(* CODESYS project RML AOIs.library
   Title: RML AOIs
   Version: 1.1
   Placeholder: RML AOIs
   Company: RML Toolbox

Project tree, tasks and I/O mapping:
  libraries: Tc2_Database, * (Beckhoff Automation GmbH); Tc2_Drive, * (Beckhoff Automation GmbH); Tc2_EtherCAT, * (Beckhoff Automation GmbH); Tc2_IoFunctions, * (Beckhoff Automation GmbH); Tc2_MC2, * (Beckhoff Automation GmbH); Tc2_MC2_Drive, * (Beckhoff Automation GmbH); Tc2_NCI, * (Beckhoff Automation GmbH); Tc2_Standard, * (Beckhoff Automation GmbH); Tc2_SUPS, * (Beckhoff Automation GmbH); Tc2_System, * (Beckhoff Automation GmbH); Tc2_TcpIp, * (Beckhoff Automation GmbH); Tc2_Utilities, * (Beckhoff Automation GmbH); Tc3_EventLogger, * (Beckhoff Automation GmbH); Tc3_Module, * (Beckhoff Automation GmbH); Tc2_CncHli, * (Beckhoff Automation GmbH); Tc3_CNC, * (Beckhoff Automation GmbH); Tc3_CNC_Drive, * (Beckhoff Automation GmbH)
  Objects/
    F_ImplicitChecks_V4_00/
      function F_CheckDivDint [ST]
      function F_CheckDivInt [ST]
      function F_CheckDivReal [ST]
      function F_CheckIndexBounds [ST]
      function F_CheckIndexBounds_DINT [ST]
      function F_CheckIndexBounds_REAL [ST]
      function F_CheckIndexBounds_UINT [ST]
      function F_LIMIT [ST]
    FB_AnalogueInput_V4_01/
      data type E_AInputTypeConfig
      function block FB_AnalogueInput [ST]: Alarm, AlarmMute, DebounceOff_ET, DebounceOff_PT, DebounceOn_ET, DebounceOn_PT, Description, FallingEdge, Fault, FaultTimer_ET, FaultTimer_PT, ForceOn, Input, Input2, M_AlarmMonitor, M_Alarms, M_Output, M_TypeConfig, M_UnlatchManuals, M_WarningMonitor, M_Warnings, ManOff, ManOn, ManOnQa, ManQa, Name, RisingEdge, SimInput, SimInput2, SimInputQa, StandbyReset, Value_Q, Value_Qa, Warning
    FB_AnalogueOutput_V4_01/
      data type E_AOutputTypeConfig
      function block FB_AnalogueOutput [ST]: Alarm, AlarmMute, DebounceOff_ET, DebounceOff_PT, DebounceOn_ET, DebounceOn_PT, Description, FallingEdge, Fault, FaultTimer_ET, FaultTimer_PT, ForceOn, Input, Input2, M_AlarmMonitor, M_Alarms, M_Output, M_TypeConfig, M_UnlatchManuals, M_WarningMonitor, M_Warnings, ManOff, ManOn, ManOnQa, ManQa, Name, RisingEdge, SimInput, SimInput2, SimInputQa, StandbyReset, Value_Q, Value_Qa, Warning
    FB_CNC_V1_01/
      data type E_CNC_HomingMethod
      data type E_CNC_Mode
      data type E_CNC_State
      function block FB_CNC [ST]: Alarm, AlarmMute, AutoHome, AxisEnabled, Description, Fault, FaultTimer_ET, FaultTimer_PT, FeedOverride, HandwheelSelected, Homed, M_AlarmMonitor, M_Alarms, M_AxesHandler, M_ChannelHandler, M_Homing, M_ManualMode, M_Selections, M_Spindle, M_ToolHandler, M_VariableViewer, M_WarningMonitor, M_Warnings, MachineMode, Name, ProgramEnd, ToolData, Variables, Warning
      data type ST_Handwheel
      data type ST_MachineMode
      data type ST_Position
      data type ST_Spindle
      data type ST_Tool
      data type ST_VE_CHAN0
    FB_CsvLogger_V1_01/
      function block FB_CsvLogger [ST]: Alarm, AlarmMute, Description, Enable, Fault, FaultTimer_ET, FaultTimer_PT, FB_exit, M_AlarmMonitor, M_Alarms, M_Log, M_WarningMonitor, M_Warnings, Name, Warning
    FB_Cylinder_V4_01/
      data type E_CylinderTypeConfig
      function block FB_Cylinder [ST]: Alarm, AlarmMute, AutoExtend, AutoRetract, CycleExtTime_PT, CycleRetTime_PT, Description, ExFaultTime_ET, ExFaultTime_PT, ExtendReed, ExtendReed1, ExtendSol, ForceExtend, ForceRetract, M_AlarmMonitor, M_Alarms, M_CountsReset, M_Extend, M_ExtendFault, M_ReedControl, M_ReedFault, M_Retract, M_RetractFault, M_TestCycle, M_TypeConfig, M_UnlatchManuals, M_WarningMonitor, M_Warnings, ManExtend, ManOff, ManRetract, Name, ReedFaultTime_ET, ReedFaultTime_PT, RetractReed, RetractReed1, RetractSol, RtFaultTime_ET, RtFaultTime_PT, StandbyReset, Variables, Warning
    FB_Database_V4_00/
      DUTs/
        data type ST_Example
      SQL Scripts/
        USP_Example.sql
        USP_Example_TestCall.sql
      Stored Procedures/
        function block FB_Example [ST]
      CurrentConfigDataBase.xml
      data type E_DatabaseType
      function block FB_Tc2Database [ST]: Alarm, AlarmMute, Description, M_AlarmMonitor, M_DbAlarms, M_DbServerAlarms, M_OdbcAlarms, Name
    FB_Diagnostics_V4_01/
      function block FB_Diagnostics [ST]: Alarm, AlarmMute, Description, F_DeviceState_to_String, F_LinkState_to_String, FaultTimer_PT, M_AlarmMonitor, M_AlarmReset, M_Alarms, M_CPU, M_Masters, M_Slaves, M_WarningMonitor, M_Warnings, Name, Warning
      data type ST_Diagnostics
      data type ST_MasterData
    FB_DolMotor_V4_03/
      function block FB_DolMotor [ST]: Alarm, AlarmMute, AutoFwd, AutoRev, Description, Fault, FaultTimer_PT, ForceOff, ForceOnFwd, ForceOnRev, IsolatorFeedback, M_AlarmMonitor, M_Alarms, M_MotorOutputs, M_UnlatchManuals, M_WarningMonitor, M_Warnings, ManOff, ManOnFwd, ManOnRev, ManSP1, MotorOn_ET, Name, OverloadFeedback, RunFeedback, Running, StandbyReset, StartTimer_PT, TotalMotorOnHours, TypeConfig, ValueFwd, ValueRev, Variables, Velocity, Warning
    FB_EventLogger_V4_02/
      function block FB_EventLogger [ST]: M_LogAlarm, M_LogAlert, M_LogMessage, M_LogWarning
    FB_MachineInformation_V4_00/
      function block FB_MachineInfo [ST]: M_CPU
    FB_MachinePerformance_V4_00/
      function block FB_MachinePerformance [ST]
      data type ST_Performance_SP
    FB_MiscInput_V4_02/
      data type E_InputTypeConfig
      function block FB_MiscInput [ST]: Alarm, AlarmMute, AutoStandbyReset, DebounceOff_ET, DebounceOff_PT, DebounceOn_ET, DebounceOn_PT, Description, EvaluationError, FallingEdge, Fault, FaultTimer_ET, FaultTimer_PT, ForceOn, Input, Input2, M_AlarmMonitor, M_Alarms, M_TypeConfig, M_UnlatchManuals, M_WarningMonitor, M_Warnings, ManOff, ManOn, Name, RisingEdge, SimInput, TestPulse1Fault, TestPulse2Fault, TestPulseGeneralFault, Value, Warning
    FB_MiscOutput_V4_01/
      function block FB_MiscOutput [ST]: Alarm, AlarmMute, Auto, CycleCount, Description, Fault, FaultTimer_ET, FaultTimer_PT, ForceOff, ForceOn, Input, M_AlarmMonitor, M_Alarms, M_SetOutput, M_UnlatchManuals, M_WarningMonitor, M_Warnings, ManOff, ManOn, Name, OutputOff_ET, OutputOn_ET, StandbyReset, Value, Warning
    FB_OEE_V3_01/
      function block FB_OEE [ST]
      data type ST_OEE
      data type ST_OEE_Flags_SP
      data type ST_OEE_In
      data type ST_OEE_Out
      data type ST_OEE_SP
    FB_PML_V4_01/
      function block FB_PackML [ST]: M_Administration, M_Commands, M_Indicators, M_ModeControl, M_SafetyBreach, M_StateMapping, M_StateTransitions, M_TransitionCounts
      data type ST_PMLAdmin
      data type ST_PMLControl
      data type ST_PMLData
      data type ST_PMLIndicators
      data type ST_PMLModualCommands
      data type ST_PMLState
      data type ST_PMLStatus
    FB_Service_V3_00/
      function block FB_Service [ST]
    FB_Servo_V4_07/
      Helpers/
        function F_ServoCheckWindow [ST]
        function F_ServoDirection [ST]
        function F_ServoPositionCheck [ST]
        function block FB_ServoMotionDynamics [ST]
        function block FB_ServoMove [LD]
      data type E_MoveState
      data type E_ServoMoveType
      function block FB_Servo [ST]: Alarm, AlarmMute, AutoEn, AutoHome, AxisEnabled, CamInSync, ContinuousRun, ContRun, Description, DigitalInputs, ExtControl, ExtManEn, Fault, FaultTimer_ET, FaultTimer_PT, ForceNeg, ForcePos, Homed, HomeMode, Jog, M_AlarmMonitor, M_Alarms, M_BrakeControl, M_ContinuousRun, M_ControlOutputs, M_Errors, M_GetDiagnosis, M_Homing, M_Jogging, M_MotionDynamicMove, M_MoveSuperImposed, M_MoveToPosition, M_SettingsControl, M_StateControl, M_StateOutputs, M_UnlatchManuals, M_WarningMonitor, M_Warnings, ManBrakeRelease, ManEn, ManHome, MoveDynamic, MovePos, MovePosSync, MoveSuperImpose, Moving, Name, PosDynamicOK, PosMove, PosMoveHome, PosOK, PosSyncOK, RunCam, StandStill, Unit, Variables, Warning
      data type ST_CamTable
      data type ST_ConstantVelocity_SP
      data type ST_HomePosition_SP
      data type ST_MovePosition_SP
      data type ST_MoveSuperImposed_SP
      data type ST_Settings_SP
    FB_Statistics_V4_02/
      function block FB_Statistics [ST]: CurrentRate, CycleTime, History, HistoryAvg, InstHistory, LastHour, LastMin, Reset, ThisHour, ThisMin
    FB_StepEngine_V4_03/
      function block FB_StepEngine [ST]: Alarm, AlarmMute, CurrentStep, Description, DeviceAlarm, Disable, Disabled, Fault, History, LastActiveStep, M_AlarmMonitor, M_Alarms, Name, SeqInterface, StepNum, StepReq, StepTime_ET, StepTimeDn, Variables
      data type ST_SequenceHistory
      data type ST_SequenceInterface
    FB_SystemEvent_V4_00/
      data type E_EventType
      function block FB_SystemEvent [ST]: Alarm, AlarmMute, EventTimer_ET, EventTimer_PT, Warning
    FB_TcpIpClient_V4_01/
      Example Server/
        TcpIp Sample.ivs
      data type E_ClientDataExchangeSteps
      data type E_ConnectionSteps
      function block FB_TcpIpClient [ST]: Alarm, AlarmMute, Description, Fault, FaultTimer_PT, M_AlarmMonitor, M_Alarms, M_DataExchange, M_Errors, M_MessageMonitor, M_Messages, M_WarningMonitor, M_Warnings, Name, Warning
    FB_TcpIpServer_V4_00/
      Example Client/
        EIO.cfg
        Rapid.mod
      data type E_ClientSteps
      data type E_ServerDataExchangeSteps
      data type E_ServerSteps
      function block FB_TcpIpServer [ST]: Alarm, AlarmMute, Description, Fault, FaultTimer_PT, M_AlarmMonitor, M_Alarms, M_DataExchange, M_Errors, M_MessageMonitor, M_Messages, M_RemoteClient, M_WarningMonitor, M_Warnings, Name, Warning
    FB_TimeManagement_V4_00/
      function block FB_TimeManagement [ST]: A_FirstCycle, A_LastScanTime, A_Strobes, A_SyncSystemTime, A_TimePulses, A_UpTime
      data type ST_ElapsedTime
      data type ST_TimeManagement
      data type ST_TimeManagement_SP
    FB_TwinSAFE_V4_01/
      function block FB_TwinSAFE [ST]: Alarm, Description, FaultTimer_ET, FaultTimer_PT, M_AlarmMonitor, M_Alarms, M_Control, M_WarningMonitor, M_Warnings, Name, Warning
    System_V4_01/
      data type ST_Selection
      data type ST_System
      data type ST_System_In
      data type ST_System_Out
      data type ST_System_SP
      data type ST_Variable
    text list GlobalTextList
  00000000-0000-0000-0000-000000000000|Objects\FB_Database_V4_00\SQL Scripts\USP_Example.sql
  00000000-0000-0000-0000-000000000000|Objects\FB_Database_V4_00\SQL Scripts\USP_Example_TestCall.sql
  00000000-0000-0000-0000-000000000000|Objects\FB_Database_V4_00\CurrentConfigDataBase.xml
  00000000-0000-0000-0000-000000000000|Objects\FB_TcpIpClient_V4_01\Example Server\TcpIp Sample.ivs
  00000000-0000-0000-0000-000000000000|Objects\FB_TcpIpServer_V4_00\Example Client\EIO.cfg
  00000000-0000-0000-0000-000000000000|Objects\FB_TcpIpServer_V4_00\Example Client\Rapid.mod
*)

// Objects/FB_AnalogueInput_V4_01/E_AInputTypeConfig
TYPE E_AInputTypeConfig :(
(*Type Configuration of Input*)
	eAInputType_PLC_NO				:=  0,
	eAInputType_PLC_NC 				:=  1,
	eAInputType_SAFE_NO 			:=  2,
	eAInputType_SAFE_NC				:=  3
);
END_TYPE

// Objects/FB_AnalogueOutput_V4_01/E_AOutputTypeConfig
TYPE E_AOutputTypeConfig :(
(*Type Configuration of Input*)
	eAOutputType_PLC_NO				:=  0,
	eAOutputType_PLC_NC 			:=  1,
	eAOutputType_SAFE_NO 			:=  2,
	eAOutputType_SAFE_NC			:=  3
);
END_TYPE

// Objects/FB_CNC_V1_01/E_CNC_HomingMethod
{attribute 'qualified_only'}
{attribute 'strict'}
TYPE E_CNC_HomingMethod :
(
	Homing		:=  0,
	Measurment	:=  1
)USINT;
END_TYPE

// Objects/FB_CNC_V1_01/E_CNC_Mode
TYPE E_CNC_Mode :(
		STANDBY_MODE		:=  1,
		AUTOMATIC_MODE 		:=  2,
		MDI_MODE	 		:=  3,
		MANUAL_MODE			:=  4,
		REFERENCE_MODE		:=  5
)UDINT;
END_TYPE

// Objects/FB_CNC_V1_01/E_CNC_State
TYPE E_CNC_State :(
	DESELECTED		:=  1,
	SELECTED 		:=  2,
	READY	 		:=  3,
	ACTIVE			:=  4,
	HOLD			:=  5,
	ERROR			:=  6,
	SELECTING		:=  7,
	DESELECTING		:=  8,
	PREPARING		:=  9,
	CLEARING		:=  10,
	STARTING		:=  11,
	ABORTING		:=  12,
	STOPPING		:=  13,
	RESUMING		:=  14,
	RESETTING		:=  15
)UDINT;
END_TYPE

// Objects/FB_CNC_V1_01/ST_Handwheel
TYPE ST_Handwheel :
STRUCT
	xAxisSelect		AT %I*		: BOOL;
	yAxisSelect		AT %I*		: BOOL;
	zAxisSelect		AT %I*		: BOOL;
	aAxisSelect		AT %I*		: BOOL;
	cAxisSelect		AT %I*		: BOOL;
	x10Resolution	AT %I*		: BOOL;
	x100Resolution	AT %I*		: BOOL;
	Handwheel 		AT %I*		: UINT;		//Increments for handwheel e.g. EL5101
END_STRUCT
END_TYPE

// Objects/FB_CNC_V1_01/ST_MachineMode
TYPE ST_MachineMode :
STRUCT
	/// Operation Mode 
	Standby: BOOL;
	Manual: BOOL;
	MDI: BOOL;
	Automatic: BOOL;
	Homing: BOOL;
	Select : BOOL; 
	Ready  : BOOL;
	Start: BOOL;
	Stop: BOOL;
	Reset: BOOL;
	Error: BOOL;
	Mode: UDINT;
	State: UDINT;
	/// Special functions 
	ChannelSignals: ST_ChannelSignals;
	BlockSearch: ST_BlockSearch;
	SyntaxCheck: ST_SyntaxCheck;
	ManualMode: ST_ManualMode;
	/// Strings 
	ProgramName: STRING(1024);
	MDIString: STRING(1024);
END_STRUCT
END_TYPE

// Objects/FB_CNC_V1_01/ST_Position
TYPE ST_Position :
STRUCT
	X	:	LREAL;
	Y	: 	LREAL;
	Z	: 	LREAL;
	C	: 	LREAL;
	A	: 	LREAL;
	rotX: 	LREAL;
	rotY: 	LREAL;
	rotZ: 	LREAL;
END_STRUCT
END_TYPE

// Objects/FB_CNC_V1_01/ST_Spindle
TYPE ST_Spindle :
STRUCT
	M3				: BOOL;			//Rotate Clockwise
	M4				: BOOL;			//Rotate Counter-Clockwise
	M5				: BOOL;			//Stop Spindle
	M7				: BOOL;			//Close Tool Holder
	M8				: BOOL;			//Tool Release
	M9				: BOOL;			//Tool Engage
	M19				: BOOL;			//Position Spindle (Closed-loop positioning only)
	ComVelocity		: DINT;			//Command Velocity
	ActVelocity		: LREAL;		//Actual Velocity
	Position		: DINT;			//Position Feedback
	Error			: BOOL;			//Error State
	ErrorID			: UDINT;		//Error ID
	Warm			: BOOL;			//Spindle is Warm
END_STRUCT
END_TYPE

// Objects/FB_CNC_V1_01/ST_Tool
TYPE ST_Tool :
STRUCT
	Desc	:	STRING;			// Tool Description
	Length	:	LREAL;			// Tool Length from Spindle Flange
	X		:	LREAL;			// X Location in Machine Coordinates
	Y		: 	LREAL;			// Y Location in Machine Coordinates
	Z		: 	LREAL;			// Z Location in Machine Coordinates
	SafeX	: 	LREAL;			// Safe X Location in Machine Coordinates
END_STRUCT
END_TYPE

// Objects/FB_CNC_V1_01/ST_VE_CHAN0
TYPE ST_VE_CHAN0 :
STRUCT
	Name			: STRING[127];
	Table 			: ST_Position;
	TableHeight		: LREAL;
	ParkPos 		: ST_Position;
END_STRUCT
END_TYPE

// Objects/FB_Cylinder_V4_01/E_CylinderTypeConfig
TYPE E_CylinderTypeConfig :(
(*Type Configuration of Cylinder*)
	eCylinderType_SINGLE_NORMAL			:=  0,
	eCylinderType_SINGLE_REVERSE 		:=  1,
	eCylinderType_DUEL 					:=  2
);
END_TYPE

// Objects/FB_Database_V4_00/DUTs/ST_Example
TYPE ST_Example :
STRUCT
	TimeStamp	   					:			STRING(31);//Time of Check
	UID	  							:			STRING(31);//8 Byte Unique Mac Id
	DataOk							:			STRING(31);//0=Fail, 1=Pass, 2=NA
	VisionOk						:			STRING(31);//0=Fail, 1=Pass, 2=NA
	VisionCause						:			STRING(31);//Cause of Vision Failure if Applicable
	VisionScore						: 			USINT;//0-100% Tag Find Score	
	Cycles							: 			USINT;//Amount of Cycles Through Machine
	Age	   							:			STRING(31);//Age of Tag
END_STRUCT
END_TYPE

// Objects/FB_Database_V4_00/E_DatabaseType
TYPE E_DatabaseType :(
	eMicrosoftSqlCompact				:=  0,
	eMicrosoftSql						:=  1,
	eMicrosoftAccess 					:=  2,
	eMySQL								:=  3,
	eOracle 							:=  4,
	eDB2								:=  5,
	ePostgreSQL							:=  6,
	eInterbase 							:=  7,
	eXml								:=  8,
	eAscii								:=  10
);
END_TYPE

// Objects/FB_Diagnostics_V4_01/ST_Diagnostics
TYPE ST_Diagnostics :
STRUCT
	Name					: STRING;
	ProductType				: STRING;
	CRCError				: DWORD;
	Address					: WORD;
	LinkStatus				: STRING;
	DeviceStatus			: STRING;
	NetId					: T_AmsNetId;
	LostFrames     			: UDINT;
	FramesPerSecond        	: LREAL;
	LostQueuedFrames      	: UDINT;
	QueuedFramesPerSecond 	: LREAL;
END_STRUCT
END_TYPE

// Objects/FB_Diagnostics_V4_01/ST_MasterData
TYPE ST_MasterData :
STRUCT
	ID						: WORD;
	Name					: STRING;
	Status					: STRING;
	NetId					: T_AmsNetId;
	LostFrames     			: UDINT;
	FramesPerSecond        	: LREAL;
	LostQueuedFrames      	: UDINT;
	QueuedFramesPerSecond 	: LREAL;
END_STRUCT
END_TYPE

// Objects/FB_MachinePerformance_V4_00/ST_Performance_SP
TYPE ST_Performance_SP :
STRUCT
	Current_Time							: DINT;
	Current									: ST_TIMEMANAGEMENT;
	Today_Time								: DINT;
	Today									: ST_TIMEMANAGEMENT;
	Today_Freq								: DINT;
	Today_Percent							: REAL;
	LifeTime_Time							: DINT;
	LifeTime								: ST_TIMEMANAGEMENT;
	LifeTime_Freq							: DINT;
	LifeTime_Percent						: REAL;	
END_STRUCT
END_TYPE

// Objects/FB_MiscInput_V4_02/E_InputTypeConfig
TYPE E_InputTypeConfig :(
(*Type Configuration of Input*)
	eInputType_PLC_NO				:=  0,
	eInputType_PLC_NC 				:=  1,
	eInputType_SAFE_NO 				:=  2,
	eInputType_SAFE_NC				:=  3,
	eInputType_SAFE_DUAL_NO 		:=  4,
	eInputType_SAFE_DUAL_NC 		:=  5,
	eInputType_SAFE_DUAL_NO_NC		:=  6
);
END_TYPE

// Objects/FB_OEE_V3_01/ST_OEE
TYPE ST_OEE :
STRUCT
	Inputs										: ST_OEE_In;
	Outputs										: ST_OEE_Out;
END_STRUCT
END_TYPE

// Objects/FB_OEE_V3_01/ST_OEE_Flags_SP
TYPE ST_OEE_Flags_SP :
STRUCT
	InfeedNotOK							: BOOL;				//Infeed supply below machine specification rate
	OutfeedNotOK						: BOOL;				//Dwnstreem equipment is stopping the machine from running
	GoodPiece							: BOOL;				//Good product
	RejectPiece							: BOOL;				//Reject Product
	BreakActive							: BOOL;				//Break active has been selected
	GoodPiece_Increment					: DINT;				//Good piece increment rate
	RejectPiece_Increment				: INT;				//Reject piece increment rate
	TargetProductRate					: REAL;				//Target Product Rate Per Minute
	TargetBoxRate						: REAL;				//Target Box Rate Per Minute
	BreakActive_ALM						: BOOL; 		    //Break active alarm
	InfeedTimer							: TON;				//Infeed Availability Timer
	OutfeedTimer						: TON;				//Outfeed Availability Timer
END_STRUCT
END_TYPE

// Objects/FB_OEE_V3_01/ST_OEE_In
TYPE ST_OEE_In :
STRUCT
	Sec_PulseTrigger										: BOOL;
	Break_Active											: BOOL;
	EnableIn												: BOOL;	
	Select													: BOOL;
END_STRUCT
END_TYPE

// Objects/FB_OEE_V3_01/ST_OEE_Out
TYPE ST_OEE_Out :
STRUCT
	Quality												: REAL;
	Performance											: REAL;
	Availability										: REAL;
	OEE													: REAL;
	Active												: BOOL;
	EnableOut											: BOOL;	
END_STRUCT
END_TYPE

// Objects/FB_OEE_V3_01/ST_OEE_SP
TYPE ST_OEE_SP :
STRUCT
	Start								: ST_TimeManagement;
	Stop								: ST_TimeManagement;
	Length								: ST_TimeManagement;
	Operating_Time						: ST_TimeManagement;
	Production_Time						: ST_TimeManagement;
	Break_Time							: ST_TimeManagement;
	SupplyDownTime_Time					: ST_TimeManagement;
	OutfeedDownTime_Time				: ST_TimeManagement;
	DownTime_Time						: ST_TimeManagement;			
	StartConcate						: LINT;
	StopConcate							: LINT;
	Active								: BOOL;
	ONS									: DINT;
	Operating_Seconds					: REAL;
	Production_Seconds					: REAL;
	Planned_Production					: DINT;
	StartStopConcate_Update				: BOOL;
	Break_Active						: BOOL;
	Break_Seconds						: DINT;
	TargetRate							: REAL;
	GoodPieces							: DINT;
	RejectPieces						: DINT;
	TotalPieces							: DINT;
	Availability						: REAL;
	Performance							: REAL;
	Quality								: REAL;
	OEE									: REAL;
	StateCurrent						: DINT;		
	MachinePerformance					: ARRAY[0..18] OF  ST_Performance_SP;
	SupplyDownTime_Seconds		 		: REAL;
	SupplyAvaliability					: REAL;
	OutfeedDownTime_Seconds				: REAL;
	OutfeedAvaliability					: REAL;
	DownTime_Seconds					: DINT;
	ShiftName							: STRING[22];
	RisingEdge							: BOOL;
END_STRUCT
END_TYPE

// Objects/FB_PML_V4_01/ST_PMLAdmin
TYPE ST_PMLAdmin :
STRUCT
	ModeCurrentTime				: ARRAY[0..7] OF DINT;				//Time spent in Mode
	ModeCummulativeTime			: ARRAY[0..7] OF DINT;				//Cumulative Time In Each Mode
	StateCurrentTime			: ARRAY[0..7,0..17] OF DINT;		//Value of last State Timer in each [mode].State[#]
	StateCummulativeTime		: ARRAY[0..7,0..17] OF DINT;		//Cumulative Time In Each [mode].State[#]
	ProdProcessed				: DINT;								//Number Products Processed
	DefectProd					: DINT;								//Number Defective Products
	StopReason					: DINT;								//The stop reason is the first event captured during an abort, held, suspended or stop event.
	ReworkProd					: DINT;								//Number Re-workable Products
	ResetTimerCounters			: BOOL;								//Reset timers and counters
END_STRUCT
END_TYPE

// Objects/FB_PML_V4_01/ST_PMLControl
TYPE ST_PMLControl :
STRUCT
	UnitMode					: DINT := 1;				//Unit Mode Target
	UnitModeChangeRequest		: BOOL;						//Request Unit Mode Change
	CurMachSpeed				: REAL;						//Current Machine Speed
	MatReady					: ARRAY[0..31] OF BOOL;		//Materials Ready
	MatLow						: ARRAY[0..31] OF BOOL;		//Materials Low
	State						: DINT;						//Target State
	StateChangeRequest			: BOOL;						//State Change Request
	CntrlCmd					: DINT;						//Control Command
	EquipmentInterLockBlocked 	: BOOL;						//Indicates that a downstream system is not able to accept product
	EquipmentInterLockStarved	: BOOL;						//Indicates that an upstream system is not able to supply product
END_STRUCT
END_TYPE

// Objects/FB_PML_V4_01/ST_PMLData
TYPE ST_PMLData :
STRUCT
	Control						: ST_PMLControl;						//PackML control data
	Status						: ST_PMLStatus;							//PackML status data
	Admin						: ST_PMLAdmin;							//PackML administration Data
	StateCtrl					: ST_PMLModualCommands;					//PackML state control commands
	Indicator					: ST_PMLIndicators;						//PackML interfaces
END_STRUCT
END_TYPE

// Objects/FB_PML_V4_01/ST_PMLIndicators
TYPE ST_PMLIndicators :
STRUCT
	LS_H_Output					: DINT;								//Matrix Output
	RedLamp						: BOOL;								//Red Lamp
	AmberLamp					: BOOL;								//Amber Lamp
	BlueLamp					: BOOL;								//Blue Lamp
	GreenLamp					: BOOL;								//Green Lamp
	PB_Output					: DINT;								//Matrix Output
	RedButton					: BOOL;								//Red Button 
	AmberButton					: BOOL;								//Amber Button 
	BlueButton					: BOOL;								//Blue Button 
	GreenButton					: BOOL;								//Green Button 
	Horn						: BOOL;								//Horn
END_STRUCT
END_TYPE

// Objects/FB_PML_V4_01/ST_PMLModualCommands
TYPE ST_PMLModualCommands :
STRUCT
	Cmd_Reset				: BOOL;			//Reset
	Sts_Resetting_SC		: BOOL;			//Resetting State Complete
	Cmd_Start				: BOOL;			//Start
	Sts_Starting_SC			: BOOL;			//Starting State Complete
	Cmd_Stop				: BOOL;			//Stop
	Sts_Stopping_SC			: BOOL;			//Stopping State Complete
	Cmd_Hold				: BOOL;			//Hold
	Sts_Holding_SC			: BOOL;			//Holding State Complete
	Cmd_UnHold				: BOOL;			//UnHold
	Sts_UnHolding_SC		: BOOL;			//UnHolding State Complete
	Cmd_Suspend				: BOOL;			//Suspend
	Sts_Suspending_SC		: BOOL;			//Suspending State Complete
	Cmd_UnSuspend			: BOOL;			//UnSuspend
	Sts_UnSuspending_SC		: BOOL;			//UnSuspending State Complete
	Cmd_Abort				: BOOL;			//Abort
	Sts_Aborting_SC			: BOOL;			//Aborting State Complete
	Cmd_Clear				: BOOL;			//Clear
	Sts_Clearing_SC			: BOOL;			//Clearing State Complete
	Sts_Execute_SC			: BOOL;			//Execute State Complete
	Sts_Completing_SC		: BOOL;			//Completing State Complete
END_STRUCT
END_TYPE

// Objects/FB_PML_V4_01/ST_PMLState
TYPE ST_PMLState :
STRUCT
	CurrentState		: DINT;
	Clearing			: BOOL;
	Stopped				: BOOL;
	Starting			: BOOL;
	Idle				: BOOL;
	Suspended			: BOOL;
	Execute				: BOOL;
	Stopping			: BOOL;
	Aborting			: BOOL;
	Aborted				: BOOL;
	Holding				: BOOL;
	Held				: BOOL;
	UnHolding			: BOOL;
	Suspending			: BOOL;
	UnSuspending		: BOOL;
	Resetting 			: BOOL;
	Completing			: BOOL;
	Complete			: BOOL;
END_STRUCT
END_TYPE

// Objects/FB_PML_V4_01/ST_PMLStatus
TYPE ST_PMLStatus :
STRUCT
	CommandRejected							: BOOL;							//Command Rejected
	UnitModeCurrent							: DINT;							//0 = Invalid, 1 = Production, 2 = Maintenance, 3 = Manual, 4 = Batch Production
	UnitModeRequested						: BOOL;							//Requested Unit Mode Change
	UnitModeChangeInProcess					: BOOL;							//Requested Unit Mode Change In Progress
	StateCurrent				AT	%Q*		: DINT;							//Current State Number
	StateRequested							: DINT;							//Target State
	StateChangeInProgress					: BOOL;							//State Change in Progress
	StateChangeProgress						: DINT;							//Percent Complete
	StateLastCompleted						: DINT;							//Last Completed State
	SeqNumber								: DINT;							//Pack ML Sequence Number
	CurMachspd								: DINT;							//Pack ML Current Machine Speed
	MatReady								: ARRAY[0..31] OF BOOL;			//Material Ready
	MatLow									: ARRAY[0..31] OF BOOL;			//Material Ready or Low
	MachDesignSpeed							: REAL;							//Machine Design Speed
	MachCycle								: DINT;							//Machine Cycle Count
	ProdRatio								: DINT;							//Count of primary packages per secondary package
	Dirty									: BOOL;							//Dirty indicator
	Clean									: BOOL;							//Clean indicator
	TimeToDirty								: DINT;							//Time remaining
	EquipmentAllocatedToUnitModeID			: DINT;							//Machinery Unit mode allocation
	MachineReusableForUnitModeID			: DINT;							//Resuable Unit Mode ID
	MachineReusableTimeLeft					: DINT;							//Reusable Time
	MachineStoringProductID					: DINT;							//Storing Product ID
	MachineTransferringProductID			: DINT;							//Transferring Product ID
	EquipmentInterLockBlocked 				: BOOL;							//Indicates that a downstream system is not able to accept product
	EquipmentInterLockStarved				: BOOL;							//Indicates that an upstream system is not able to supply product
END_STRUCT
END_TYPE

// Objects/FB_Servo_V4_07/E_MoveState
TYPE E_MoveState :
(
	MOVESTATE_INIT,
	MOVESTATE_ENABLE,
	MOVESTATE_FORWARD,
	MOVESTATE_BACKWARDS,
	MOVESTATE_BACKWARDSSLOW,
	MOVESTATE_NEWTARGETPOSITION,
	MOVESTATE_ERROR,
	MOVESTATE_RESET,
	MOVESTATE_CAMIN,
	MOVESTATE_SWITCHCAM,
	MOVESTATE_READCAMDATA,
	MOVESTATE_PREPARECAMMODIFICATION,
	MOVESTATE_MODIFYCAM,
	MOVESTATE_CAMSCALING,
	MOVESTATE_CAMOUT,
	MOVESTATE_STOPMASTER,
	MOVESTATE_STOPAXES
);
END_TYPE

// Objects/FB_Servo_V4_07/E_ServoMoveType
TYPE E_ServoMoveType :(
	(*Move Type Configuration of Positional Move*)
	eServoMoveType_ABSOLUTE							:=  0,
	eServoMoveType_RELATIVE 						:=  1,
	eServoMoveType_MODULO_SHORTEST_PATH 			:=  2,
	eServoMoveType_MODULO_POSITIVE 					:=  3,
	eServoMoveType_MODULO_NEGATIVE					:=  4,
	eServoMoveType_ABSOLUTE_MASTER_OFFSET 			:=  5,
	eServoMoveType_INCREMENTAL_MASTER_OFFSET		:=  6
);
END_TYPE

// Objects/FB_Servo_V4_07/ST_CamTable
TYPE ST_CamTable :
STRUCT
	TableData 		: ARRAY [0..360,0..1] OF LREAL;
	Id				: UDINT;
	Rows			: UDINT;
	Periodic		: BOOL;
	Generate		: BOOL;
	//StartMode		: MC_StartMode;
END_STRUCT
END_TYPE

// Objects/FB_Servo_V4_07/ST_ConstantVelocity_SP
TYPE ST_ConstantVelocity_SP :
STRUCT
	Direction			: MC_Direction;			//Direction of Constant Move
	Velocity			: REAL := 50;			//Velocity Value of Move
	Acceleration		: REAL := 1;			//Accleration Value of Move
	Deceleration		: REAL := 1;			//Deceleration Value of Move
	Jerk				: REAL :=25;			//Jerk Value of Move
END_STRUCT
END_TYPE

// Objects/FB_Servo_V4_07/ST_HomePosition_SP
TYPE ST_HomePosition_SP :
STRUCT
	Position			: REAL;					//Position Value to Move to
	FastVelocity		: REAL := 50;			//Fast Velocity Value of Move
	SlowVelocity		: REAL := 10;			//Slow Velocity Value of Move
	Acceleration		: REAL := 10000;		//Accleration Value of Move
	Deceleration		: REAL := 10000;		//Deceleration Value of Move
	Jerk				: REAL := 10000;		//Jerk Value of Move
	Timeout				: REAL := 5;			//Time Allowed for Move to Complete
END_STRUCT
END_TYPE

// Objects/FB_Servo_V4_07/ST_MovePosition_SP
TYPE ST_MovePosition_SP :
STRUCT
	MoveType			: E_ServoMoveType;		//Move Type Configuration of Positional Move
	Position			: REAL;					//Position Value to Move to
	Velocity			: REAL := 50;			//Velocity Value of Move
	Acceleration		: REAL := 1;			//Accleration Value of Move
	Deceleration		: REAL := 1;			//Deceleration Value of Move
	Jerk				: REAL := 25;			//Jerk Value of Move
	Timeout				: REAL := 5;			//Time Allowed for Move to Complete
END_STRUCT
END_TYPE

// Objects/FB_Servo_V4_07/ST_MoveSuperImposed_SP
TYPE ST_MoveSuperImposed_SP :
STRUCT
	Distance			: REAL;					//Relative distance to catch up or fall back with the super imposed move
	Velocity			: REAL := 50;			//Velocity Value of Move without move super imposed
	VelocityDiff		: REAL := 50;			//Velocity Value of the catch up or fall back distance
	Acceleration		: REAL := 1;			//Accleration Value of Move
	Deceleration		: REAL := 1;			//Deceleration Value of Move
	Length				: REAL;					//Length of the total move distance
END_STRUCT
END_TYPE

// Objects/FB_Servo_V4_07/ST_Settings_SP
TYPE ST_Settings_SP :
STRUCT
	HomeOffsetPosition			: LREAL;			//Home Offset Position
	HomeRequired				: BOOL;				//Used if Servo is Homed from Marker
	MaxPositionLag				: LREAL;			//Maximum Position Lag Value
	MaxPositionLagTime			: LREAL;			//Filter Time for Maximum Position Lag
	SoftPositionLimitMaxActive	: BOOL;				//Activates Soft Position Maximum Limit Monitoring
	SoftPositionLimitMinActive	: BOOL;				//Activates Soft Position Minimum Limit Monitoring
	SoftPositionLimitMax		: LREAL;			//Maximum Soft Position Limit
	SoftPositionLimitMin		: LREAL;			//Minimum Soft Position Limit
	PositionTollerance			: REAL := 1;		//Window for position OK
	ModuloFactor				: LREAL;			//Modulo (unwind) value read form drive parameters
	HomingCamSearchDirection	: BOOL;				//Direction for homing drive
	HomingSyncSearchDirection	: BOOL;				//Direction for second stage of homing
END_STRUCT
END_TYPE

// Objects/FB_StepEngine_V4_03/ST_SequenceHistory
TYPE ST_SequenceHistory :
STRUCT
	StepNum			: INT;
	StepTime		: REAL;
	Message 		: STRING; 
END_STRUCT
END_TYPE

// Objects/FB_StepEngine_V4_03/ST_SequenceInterface
TYPE ST_SequenceInterface :
STRUCT
	Held					: BOOL;
	Stopped					: BOOL;
	Reset					: BOOL;
	Suspended				: BOOL;
	Complete				: BOOL;
END_STRUCT
END_TYPE

// Objects/FB_SystemEvent_V4_00/E_EventType
TYPE E_EventType :(
	eAlarm							:=  0,
	eWarning		 				:=  1,
	eAlert		 					:=  2,
	eMessage		 				:=  3
)USINT;
END_TYPE

// Objects/FB_TcpIpClient_V4_01/E_ClientDataExchangeSteps
TYPE E_ClientDataExchangeSteps :
(
	CLIENT_DATAEXCHANGE_STATE_IDLE,
	CLIENT_DATAEXCHANGE_STATE_SEND_START,
	CLIENT_DATAEXCHANGE_STATE_SEND_WAIT,
	CLIENT_DATAEXCHANGE_STATE_RECEIVE_START,
	CLIENT_DATAEXCHANGE_STATE_RECEIVE_WAIT,
	CLIENT_DATAEXCHANGE_STATE_ERROR
);
END_TYPE

// Objects/FB_TcpIpClient_V4_01/E_ConnectionSteps
TYPE E_ConnectionSteps :
(
	CONNECTION_STATE_IDLE,
	CONNECTION_STATE_CONNECT_START,
	CONNECTION_STATE_CONNECT_WAIT,
	CONNECTION_STATE_DATAEXCHANGE_START,
	CONNECTION_STATE_DATAEXCHANGE_WAIT,
	CONNECTION_STATE_CLOSE_START,
	CONNECTION_STATE_CLOSE_WAIT,
	CONNECTION_STATE_ERROR
);
END_TYPE

// Objects/FB_TcpIpServer_V4_00/E_ClientSteps
TYPE E_ClientSteps :
(
	CLIENT_STATE_IDLE,
	CLIENT_STATE_CONNECT_START,
	CLIENT_STATE_CONNECT_WAIT,
	CLIENT_STATE_DATAEXCHANGE_START,
	CLIENT_STATE_DATAEXCHANGE_WAIT,
	CLIENT_STATE_CLOSE_START,
	CLIENT_STATE_CLOSE_WAIT,
	CLIENT_STATE_ERROR
);
END_TYPE

// Objects/FB_TcpIpServer_V4_00/E_ServerDataExchangeSteps
TYPE E_ServerDataExchangeSteps :
(
	SERVER_DATAEXCHANGE_STATE_IDLE,
	SERVER_DATAEXCHANGE_STATE_SEND_START,
	SERVER_DATAEXCHANGE_STATE_SEND_WAIT,
	SERVER_DATAEXCHANGE_STATE_RECEIVE_START,
	SERVER_DATAEXCHANGE_STATE_RECEIVE_WAIT,
	SERVER_DATAEXCHANGE_STATE_ERROR
);
END_TYPE

// Objects/FB_TcpIpServer_V4_00/E_ServerSteps
TYPE E_ServerSteps :
(
	SERVER_STATE_IDLE,
	SERVER_STATE_LISTENER_OPEN_START,
	SERVER_STATE_LISTENER_OPEN_WAIT,
	SERVER_STATE_REMOTE_CLIENTS_COMM,
	SERVER_STATE_REMOTE_CLIENTS_CLOSE,
	SERVER_STATE_LISTENER_CLOSE_START,
	SERVER_STATE_LISTENER_CLOSE_WAIT,
	SERVER_STATE_ERROR
);
END_TYPE

// Objects/FB_TimeManagement_V4_00/ST_ElapsedTime
TYPE ST_ElapsedTime :
STRUCT
	Days		: INT;
	Hours		: INT;
	Minutes		: INT;
	Seconds		: INT;
END_STRUCT
END_TYPE

// Objects/FB_TimeManagement_V4_00/ST_TimeManagement
TYPE ST_TimeManagement :
STRUCT
	CurrentTime		: TIMESTRUCT;			//Current System time
	UpTime			: ST_ElapsedTime;		//Time since last reset
	SecondPulse		: BOOL;					//On for one cycle every second
	MinutePulse		: BOOL;					//On for one cycle every minute
	HourPulse		: BOOL;					//On for one cycle every hour
	MidnightPulse	: BOOL;					//On for one cycle at Midnight
	FirstCycle		: BOOL;					//True when executing first scan
	ScanTime		: REAL;					//Last scan time (Seconds)	
	SecondsNow		: DWORD;				//Current DateTime in Seconds
	SlowFlash		: BOOL;					//Slow Flash Strobe
	FastFlash		: BOOL;					//Fast Flash Strobe
	PulseFlash		: BOOL;					//Pulse Flash Strobe
END_STRUCT
END_TYPE

// Objects/FB_TimeManagement_V4_00/ST_TimeManagement_SP
TYPE ST_TimeManagement_SP :
STRUCT
	TotalUpTime				: ST_ElapsedTime;	//Total up time of System
	PreviousDay				: INT;				//Previous day, used for midnight pulse
END_STRUCT
END_TYPE

// Objects/System_V4_01/ST_Selection
TYPE ST_Selection :
STRUCT
	Select			: BOOL;
	Queued			: BOOL;
	Enabled	    	: BOOL;
	Interlock		: BOOL;
	Messages		: STRING[255];
	Description		: STRING[255];
END_STRUCT
END_TYPE

// Objects/System_V4_01/ST_System
TYPE ST_System :
STRUCT
	Inputs					: ST_System_In;			// System inputs
	Outputs					: ST_System_Out;		// System outputs
	SystemTime				: ST_TimeManagement;	// System time and pulses	
	PackMLState				: ST_PMLState;			// System PackML data
END_STRUCT
END_TYPE

// Objects/System_V4_01/ST_System_In
TYPE ST_System_In :
STRUCT
	Start					: ST_Selection;				//Machine Start selection
	Hold					: ST_Selection;				//Machine Hold selection
	Stop					: ST_Selection;				//Machine Stop selection
	Complete				: ST_Selection;				//Machine Complete selection
	SafetyReset				: ST_Selection;				//Machine Safety Reset selection
	Reset					: ST_Selection;				//Machine Reset selection
	AlarmAck				: ST_Selection;				//Machine Alarm Acknowledge selection
	Home					: ST_Selection;				//Machine Home selection
	Simulation				: ST_Selection;				//Machine Simulation selection
	RecipeLoad				: ST_Selection;				//Operator Load Recipe Selection
	RecipeSave				: ST_Selection;				//Operator Save Recipe Selection
	RecipeChanged			: ST_Selection;				//Recipe Changed Selection
	DeleteRecipe			: ST_Selection;				//Service Reset Selection
	DoorUnlock				: ST_Selection;				//Machine Gaurd Unlock Selection
	HoursReset				: BOOL;						//Resets All Motor hours, cylinder counts, machine Hours, etc...
	AlarmMuteReset			: BOOL;						//Resets Alarm Mutes for all Alarms
	GlueStandbyReset		: BOOL;						//Resets standby for all glue machines
	Exception				: __SYSTEM.ExceptionCode;	//System Exception Handler			
END_STRUCT
END_TYPE

// Objects/System_V4_01/ST_System_Out
TYPE ST_System_Out :
STRUCT
	Energized				AT %Q*	: BOOL;					//System energized
	Energized_T1					: BOOL;					//Pneumatic soft start complete
	Energized_T2					: BOOL;					//Drives power up complete
	SafetyCellBreach				: BOOL;					//Safety cell has been breached in production state
	Alert							: BOOL;					//Machine alert active
	Alarm							: BOOL;					//Machine has an alarm active
	Warning							: BOOL;					//Machine has a warning active
	Home_EN							: BOOL;					//Machine homing is enabled
	SimulationActive				: BOOL;					//Machine simulation is active
	Energized_ET					: REAL;					//Time the system has been energized
	DeEnergized_ET					: REAL;					//Time the system has been de-energized	
	AlarmMessage					: STRING;				//Active Alarm Message
	WarningMessage					: STRING;				//Active Warning Message
	InfoMessage						: STRING;				//Active Information Message
	StatusMessage					: STRING;				//Used to display machine status on HMI
	AlertMessage					: STRING;				//Used to display alert on HMI
	RecipeSaved						: BOOL;					//Recipe Saved
	RecipeLoaded					: BOOL;					//Recipe Loaded
END_STRUCT
END_TYPE

// Objects/System_V4_01/ST_System_SP
TYPE ST_System_SP:
STRUCT
	Name					: STRING[15];			// Name for HMI
	Description				: STRING[40];			// Description for HMI
	Homed					: BOOL;					// Machine homed
	Energized_T1_PT			: REAL;					// Pneumatic soft start time
	Energized_T2_PT			: REAL;					// Drives power up time
	TimeManagement			: ST_TimeManagement_SP;	// Total up time of System
	ActiveRecipe			: STRING;				// Description of active recipe
	SelectedRecipe			: STRING;				// Description of Selected Recipe on the HMI Grid
	RecipeChanged			: BOOL;					// Recipe changed, used for operator confirmation
	ActiveRecipeIndex		: UDINT;				// Index of active recipe
END_STRUCT
END_TYPE

// Objects/System_V4_01/ST_Variable
TYPE ST_Variable :
STRUCT
	Value				:REAL;
	Description			:STRING(100);
END_STRUCT
END_TYPE

// Objects/F_ImplicitChecks_V4_00/F_CheckDivDint
FUNCTION F_CheckDivDint : DINT
VAR_INPUT
	divisor: DINT;
END_VAR

IF divisor = 0 THEN
	F_CheckDivDint:=1;
ELSE
	F_CheckDivDint:=divisor;
END_IF;

END_FUNCTION

// Objects/F_ImplicitChecks_V4_00/F_CheckDivInt
FUNCTION F_CheckDivInt : INT
VAR_INPUT
	divisor: INT;
END_VAR

IF divisor = 0 THEN
	F_CheckDivInt:=1;
ELSE
	F_CheckDivInt:=divisor;
END_IF;

END_FUNCTION

// Objects/F_ImplicitChecks_V4_00/F_CheckDivReal
FUNCTION F_CheckDivReal : REAL
VAR_INPUT
	divisor: REAL;
END_VAR

IF divisor = 0 THEN
	F_CheckDivReal:=1;
ELSE
	F_CheckDivReal:=divisor;
END_IF;

END_FUNCTION

// Objects/F_ImplicitChecks_V4_00/F_CheckIndexBounds
FUNCTION F_CheckIndexBounds : INT
VAR_INPUT
	lowerbound		: 	INT;
	upperbound		:   INT;
END_VAR
VAR_IN_OUT
	index			: 	INT;
END_VAR

IF  index < lowerbound THEN
	F_CheckIndexBounds := lowerbound;
	index 		:= lowerbound;
ELSIF  index > upperbound THEN
	F_CheckIndexBounds := upperbound;
	index 		:= upperbound;
ELSE  
	F_CheckIndexBounds := index;
END_IF

END_FUNCTION

// Objects/F_ImplicitChecks_V4_00/F_CheckIndexBounds_DINT
FUNCTION F_CheckIndexBounds_DINT : DINT
VAR_INPUT
	lowerbound		: 	DINT;
	upperbound		:   DINT;
END_VAR
VAR_IN_OUT
	index			: 	DINT;
END_VAR

IF  index < lowerbound THEN
	F_CheckIndexBounds_DINT := lowerbound;
	index 		:= lowerbound;
ELSIF  index > upperbound THEN
	F_CheckIndexBounds_DINT := upperbound;
	index 		:= upperbound;
ELSE  
	F_CheckIndexBounds_DINT := index;
END_IF

END_FUNCTION

// Objects/F_ImplicitChecks_V4_00/F_CheckIndexBounds_REAL
FUNCTION F_CheckIndexBounds_REAL : REAL
VAR_INPUT
	lowerbound		: 	REAL;
	upperbound		:   REAL;
END_VAR
VAR_IN_OUT
	index			: 	REAL;
END_VAR

IF  index < lowerbound THEN
	F_CheckIndexBounds_REAL := lowerbound;
	index 		:= lowerbound;
ELSIF  index > upperbound THEN
	F_CheckIndexBounds_REAL := upperbound;
	index 		:= upperbound;
ELSE  
	F_CheckIndexBounds_REAL := index;
END_IF

END_FUNCTION

// Objects/F_ImplicitChecks_V4_00/F_CheckIndexBounds_UINT
FUNCTION F_CheckIndexBounds_UINT : UINT
VAR_INPUT
	lowerbound		: 	UINT;
	upperbound		:   UINT;
END_VAR
VAR_IN_OUT
	index			: 	UINT;
END_VAR

IF  index < lowerbound THEN
	F_CheckIndexBounds_UINT := lowerbound;
	index 		:= lowerbound;
ELSIF  index > upperbound THEN
	F_CheckIndexBounds_UINT := upperbound;
	index 		:= upperbound;
ELSE  
	F_CheckIndexBounds_UINT := index;
END_IF

END_FUNCTION

// Objects/F_ImplicitChecks_V4_00/F_LIMIT
FUNCTION F_LIMIT : BOOL
VAR_INPUT
	En			: BOOL;
	High		: LREAL;
	Value		: LREAL;
	Low			: LREAL;
END_VAR
VAR
END_VAR

IF En = TRUE AND (Low <= High AND
 (Value >= Low AND Value <= High)) OR
 (Low >= High AND
 (Value <= Low OR Value >= High)) THEN
	F_LIMIT := TRUE;
ELSE	
	F_LIMIT := FALSE;
END_IF;

END_FUNCTION

// Objects/FB_AnalogueInput_V4_01/FB_AnalogueInput
FUNCTION_BLOCK FINAL FB_AnalogueInput EXTENDS FB_EventLogger
VAR_IN_OUT
	Control					: ST_System;
END_VAR
VAR
	_Input		AT %I*		: UINT;					//Raw Input 1 - Analogue
	_Input2		AT %I*		: BOOL;					//Raw Input 2 - Digital
	_InputLimitHigh			: REAL;					//HighHigh limit of Raw Input 1
	_InputLimitLow			: REAL;					//Low limit of Raw Input 1
	_InputLimitHighHigh		: REAL;					//HighHigh limit of Raw Input 1
	_InputLimitLowLow		: REAL;					//LowLow limit of Raw Input 1
	_ManOnQa				: BOOL;					//Manual On Analogue Input
	_ManQa					: REAL;					//Manual Analogue Input
	_ManOn					: BOOL;					//Manual On
	_ManOff					: BOOL;					//Manual Off
	_ForceOn				: BOOL;					//Force On
	_ForceOff				: BOOL;					//Force Off
	_Fault					: BOOL;					//Fault
	_SimInput				: BOOL;		        	//Simulates Analogue Input
	_SimInput2				: BOOL;					//Simulates Digital Input
	_SimInputQa				: REAL;					//Value of Simulated Analogue Input
	_Value_Q	AT %Q*		: BOOL;					//Value of Input - Digital
	_Value_Qa	AT %Q*		: REAL;					//Value of Input - Analogue
	_FallingEdge			: BOOL;					//Falling Edge of Value Signal
	_RisingEdge				: BOOL;					//Raising Edge of Value Signal
	_DebounceOn_ET			: REAL;					//Debounce On Elapsed Time
	_DebounceOff_ET			: REAL;					//Debounce Off Elapsed Time
	_FaultTimer_ET			: REAL;					//Fault timer elapsed
	_Alarm					: BOOL;					//Device Alarm
	_Warning				: BOOL;					//Device Warning
	_AlarmNum				: DINT;					//Device Alarm Number
	_WarningNum				: DINT;					//Device Warning Number
	_riseEdge				: R_TRIG;				//Rising Edge Value Trigger
	_fallEdge				: F_TRIG;				//Falling Edge Value Trigger
	_Scale_Max				: REAL;					//Current Maximum (mA)
	_Scale_Min				: REAL;					//Current minimum (mA)
	_Scale_Value			: REAL;					//Current Value (mA)
	_Bit_Value				: REAL;					//Analogue Value Input
	_Bit_Max				: REAL;					//Maximum Bit Value (typically 32767)
	_Bit_Min				: REAL;					//Minimum Bit Value (typically 0)
	_Physical_Min			: REAL;					//Minimum Physical Value
	_Physical_Max			: REAL;					//Maximum Physical Value
	_ConfInput				: BOOL;					//Confirgured Input
	_DebounceOn_DN			: BOOL;					//Debounce On Timer is Done
	_DebounceOff_DN			: BOOL;					//Debounce Off Timer is Done
	_R_Trig					: ARRAY[0..9] OF R_TRIG;//Private Rising Edge Triggers
END_VAR
VAR PERSISTENT
	_Name					: STRING[15];			//Name for HMI
	_Description			: STRING[40];			//Description for HMI
	_AlarmMute				: BOOL;					//Alarm Mute
	_TypeConfig				: E_AInputTypeConfig;	//Type congifuration
	_DebounceOn_PT			: REAL;					//Debounce on timer preset time
	_DebounceOff_PT			: REAL;					//Debounce off timer preset time
	_FaultTimer_PT			: REAL;					//Fault timer preset time
	_HighAlarmLimit			: BOOL;					//Input Value is approaching the maximum operating limit.
	_LowAlarmLimit			: BOOL;					//Input Value is approaching the minimum operating limit.
	_HighHighAlarmLimit		: BOOL;					//Input Value is above  the maximum operating limit
	_LowLowAlarmLimit		: BOOL;					//Input Value is below the minimum operating limit.
	_BitValue_Max			: INT;					//Maximum Bit Value (typically 32767)
	_BitValue_Min			: INT;					//Minimum Bit Value (typically 0)
	_PhysicalValue_Min		: INT;					//Minimum Physical Value
	_PhysicalValue_Max		: INT;					//Maximum Physical Value
	_ScaleValue_Min			: INT;					//Minimum Scale Value				
	_ScaleValue_Max			: INT;					//Maximum Scale Value
END_VAR

M_TypeConfig();
M_AlarmMonitor();
M_WarningMonitor();
M_UnlatchManuals();
M_Output();

//Debounce On Timer
IF _ConfInput = TRUE AND NOT _ForceOff AND NOT _ManOff THEN
	_DebounceOn_ET := _DebounceOn_ET + Control.SystemTime.ScanTime;
	_debounceOn_DN := _DebounceOn_ET > _DebounceOn_PT;
ELSE
	_debounceOn_DN := FALSE;
END_IF
IF _debounceOn_DN OR _ForceOn OR _ManOn THEN
	_Value_Q := TRUE;
	_DebounceOff_ET := 0;
END_IF

//Debounce Off Timer
IF _ConfInput = FALSE AND NOT _ForceOn AND NOT _ManOn THEN
	_DebounceOff_ET := _DebounceOff_ET + Control.SystemTime.ScanTime;
	_debounceOff_DN := _DebounceOff_ET > _DebounceOff_PT;
ELSE
	_debounceOff_DN := FALSE;
END_IF
IF _debounceOff_DN OR _ForceOff OR _ManOff THEN
	_Value_Q:= FALSE;
	_DebounceOn_ET := 0;
END_IF

//Rising Edge Trigger 
_riseEdge(CLK := _Value_Q);
_RisingEdge := _riseEdge.Q;

//Falling Edge Trigger
_fallEdge(CLK := _Value_Q);
_FallingEdge := _fallEdge.Q;

{attribute 'monitoring' := 'variable'}
PROPERTY PUBLIC Alarm : Bool
GET
Alarm := _Alarm;
END_GET
END_PROPERTY

{attribute 'monitoring' := 'variable'}
PROPERTY PUBLIC AlarmMute : BOOL
SET
AlarmMute := _AlarmMute;
END_SET
END_PROPERTY

{attribute 'monitoring' := 'variable'}
PROPERTY PUBLIC DebounceOff_ET : real
GET
DebounceOff_ET := _DebounceOff_ET;
END_GET
END_PROPERTY

{attribute 'monitoring' := 'variable'}
PROPERTY PUBLIC DebounceOff_PT : real
GET
DebounceOff_PT := _DebounceOff_PT;
END_GET
SET
_DebounceOff_PT := DebounceOff_PT;
END_SET
END_PROPERTY

{attribute 'monitoring' := 'variable'}
PROPERTY PUBLIC DebounceOn_ET : real
GET
DebounceOn_ET := _DebounceOn_ET;
END_GET
END_PROPERTY

{attribute 'monitoring' := 'variable'}
PROPERTY PUBLIC DebounceOn_PT : real
GET
DebounceOn_PT := _DebounceOn_PT;
END_GET
SET
_DebounceOn_PT := DebounceOn_PT;
END_SET
END_PROPERTY

{attribute 'monitoring' := 'variable'}
PROPERTY PUBLIC Description : String[40]
GET
Description := _Description;
END_GET
SET
_Description := Description;
END_SET
END_PROPERTY

{attribute 'monitoring' := 'variable'}
PROPERTY PUBLIC FallingEdge : Bool
GET
FallingEdge := _FallingEdge;
END_GET
END_PROPERTY

{attribute 'monitoring' := 'variable'}
PROPERTY PUBLIC Fault : Bool
SET
_Fault := Fault;
END_SET
END_PROPERTY

{attribute 'monitoring' := 'variable'}
PROPERTY PUBLIC FaultTimer_ET : real
GET
FaultTimer_ET := _FaultTimer_ET;
END_GET
END_PROPERTY

{attribute 'monitoring' := 'variable'}
PROPERTY PUBLIC FaultTimer_PT : real
GET
FaultTimer_PT := _FaultTimer_PT;
END_GET
SET
_FaultTimer_PT := FaultTimer_PT;
END_SET
END_PROPERTY

{attribute 'monitoring' := 'variable'}
PROPERTY PUBLIC ForceOn : Bool
GET
ForceOn := _ForceOn;
END_GET
SET
_ForceOn := ForceOn;
END_SET
END_PROPERTY

{attribute 'monitoring' := 'variable'}
PROPERTY PUBLIC Input : UINT
GET
Input := _Input;
END_GET
END_PROPERTY

{attribute 'monitoring' := 'variable'}
PROPERTY PUBLIC Input2 : Bool
GET
Input2 := _Input2;
END_GET
END_PROPERTY

METHOD PRIVATE M_AlarmMonitor
VAR_INPUT
END_VAR
VAR_INST
END_VAR
VAR_INST // added by the converter: edge detectors and wires of the graphical bodies
    _w1, _w2, _w3, _w4, _w5 : BOOL;
    _rt1 : R_TRIG;
END_VAR
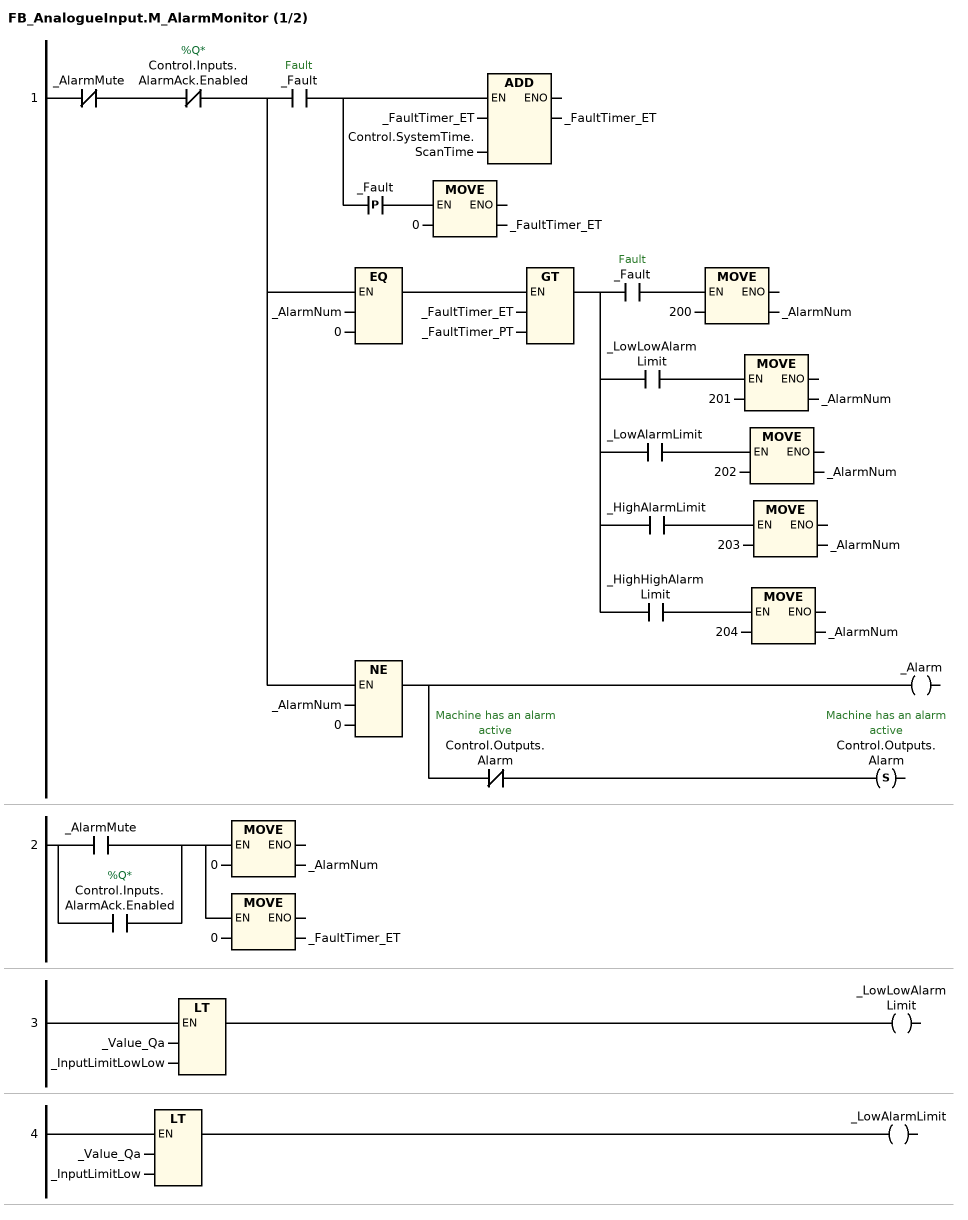
// NETWORK 1
//   Control.Inputs.AlarmAck.Enabled: AT %Q*
//   _Fault: Fault
//   _FaultTimer_ET: Fault timer elapsed
//   Control.SystemTime.ScanTime: Last scan time (Seconds)
//   _FaultTimer_PT: Fault timer preset time
//   Control.Outputs.Alarm: Machine has an alarm active
_w1 := NOT _AlarmMute AND NOT Control.Inputs.AlarmAck.Enabled;
_w2 := _w1 AND _Fault;
IF _w2 THEN _FaultTimer_ET := _FaultTimer_ET + Control.SystemTime.ScanTime; END_IF
_rt1(CLK := _Fault);
IF _w2 AND _rt1.Q THEN _FaultTimer_ET := 0; END_IF
_w3 := _w1 AND _AlarmNum = 0 AND _FaultTimer_ET > _FaultTimer_PT;
IF _w3 AND _Fault THEN _AlarmNum := 200; END_IF
IF _w3 AND _LowLowAlarmLimit THEN _AlarmNum := 201; END_IF
IF _w3 AND _LowAlarmLimit THEN _AlarmNum := 202; END_IF
IF _w3 AND _HighAlarmLimit THEN _AlarmNum := 203; END_IF
IF _w3 AND _HighHighAlarmLimit THEN _AlarmNum := 204; END_IF
_w4 := _w1 AND _AlarmNum <> 0;
_Alarm := _w4;
Control.Outputs.Alarm S= _w4 AND NOT Control.Outputs.Alarm;

// NETWORK 2
//   Control.Inputs.AlarmAck.Enabled: AT %Q*
//   _FaultTimer_ET: Fault timer elapsed
_w5 := _AlarmMute OR Control.Inputs.AlarmAck.Enabled;
IF _w5 THEN _AlarmNum := 0; END_IF
IF _w5 THEN _FaultTimer_ET := 0; END_IF

// NETWORK 3
_LowLowAlarmLimit := _Value_Qa < _InputLimitLowLow;

// NETWORK 4
_LowAlarmLimit := _Value_Qa < _InputLimitLow;

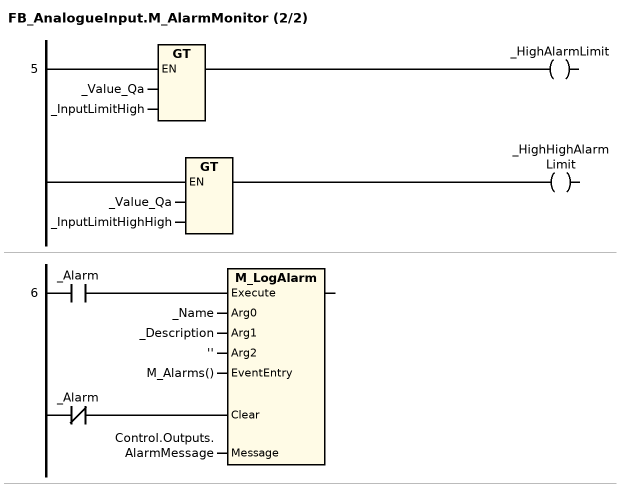
// NETWORK 5
_HighAlarmLimit := _Value_Qa > _InputLimitHigh;
_HighHighAlarmLimit := _Value_Qa > _InputLimitHighHigh;

// NETWORK 6
M_LogAlarm(Execute := _Alarm, Arg0 := _Name, Arg1 := _Description, Arg2 := '', EventEntry := M_Alarms(), Clear := NOT _Alarm, Message := Control.Outputs.AlarmMessage);
END_METHOD

METHOD PRIVATE M_Alarms : TcEventEntry
VAR_INPUT
END_VAR
CASE _AlarmNum OF
	201: M_Alarms:= TC_Events.TcAnalogueInput.A_201;//Low Low Limit Alarm
	202: M_Alarms:= TC_Events.TcAnalogueInput.A_202;//Low Limit Alarm			
	203: M_Alarms:= TC_Events.TcAnalogueInput.A_203;//High Limit Alarm
	204: M_Alarms:= TC_Events.TcAnalogueInput.A_204;//High High Limit Alarm							
ELSE
	M_Alarms:= TC_Events.TcAnalogueInput.A_Undefined;
END_CASE
END_METHOD

METHOD PRIVATE M_Output
VAR
END_VAR
VAR_INST
END_VAR
// Convert UINTs to INTs
_Scale_Min := ANY_TO_REAL(_ScaleValue_Min);
_Scale_Max := ANY_TO_REAL(_ScaleValue_Max);
_Bit_Value := ANY_TO_REAL(_Input);
_Bit_Max := ANY_TO_REAL(_BitValue_Max);		
_Bit_Min := ANY_TO_REAL(_BitValue_Min);		
_Physical_Min := ANY_TO_REAL(_PhysicalValue_Min);
_Physical_Max := ANY_TO_REAL(_PhysicalValue_Max);

IF _ManOnQa THEN
	_Value_Qa := _ManQa;
ELSIF _SimInput THEN
	_Value_Qa := _SimInputQa;
ELSIF _BitValue_Max <> 0 AND _PhysicalValue_Max <> 0 AND _ScaleValue_Max <> 0 THEN	
	// Calculate present electrical current value
	_Scale_Value := (((_Scale_Max - _Scale_Min)/F_CheckDivReal(divisor:=(_Bit_max - _Bit_min))) * (_Bit_Value - _Bit_min)) + _Scale_Min;

	// Convert electrical current value into measurable units
	_Value_Qa := (((_Physical_Max - _Physical_Min)/F_CheckDivReal(divisor:=(_Scale_Max - _Scale_Min))) * (_Scale_Value - _Scale_Min)) + _Physical_Min;	
END_IF
END_METHOD

METHOD PRIVATE M_TypeConfig
VAR_INPUT
END_VAR
VAR_INST
END_VAR
CASE _TypeConfig OF
	eAInputType_PLC_NO, eAInputType_SAFE_NO : 
		IF _Input2 OR _SimInput2 THEN
			_ConfInput := TRUE;
		ELSE
			_ConfInput := FALSE;
		END_IF
	eAInputType_PLC_NC, eAInputType_SAFE_NC : 
		IF NOT _Input2 OR _SimInput2 THEN
			_ConfInput := TRUE;
		ELSE
			_ConfInput := FALSE;
		END_IF
END_CASE
END_METHOD

METHOD PRIVATE M_UnlatchManuals
VAR_INPUT
END_VAR
VAR_INST
END_VAR
VAR_INST // added by the converter: edge detectors and wires of the graphical bodies
    _rt1, _rt2, _rt3 : R_TRIG;
END_VAR
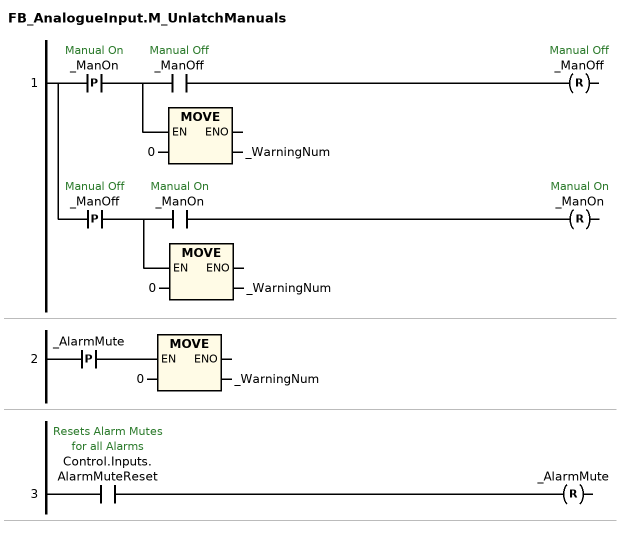
// NETWORK 1
//   _ManOn: Manual On
//   _ManOff: Manual Off
_rt1(CLK := _ManOn);
_ManOff R= _rt1.Q AND _ManOff;
IF _rt1.Q THEN _WarningNum := 0; END_IF
_rt2(CLK := _ManOff);
_ManOn R= _rt2.Q AND _ManOn;
IF _rt2.Q THEN _WarningNum := 0; END_IF

// NETWORK 2
_rt3(CLK := _AlarmMute);
IF _rt3.Q THEN _WarningNum := 0; END_IF

// NETWORK 3
//   Control.Inputs.AlarmMuteReset: Resets Alarm Mutes for all Alarms
_AlarmMute R= Control.Inputs.AlarmMuteReset;
END_METHOD

METHOD PRIVATE M_WarningMonitor
VAR_INPUT
END_VAR
VAR_INST
END_VAR
VAR_INST // added by the converter: edge detectors and wires of the graphical bodies
    _w1 : BOOL;
END_VAR
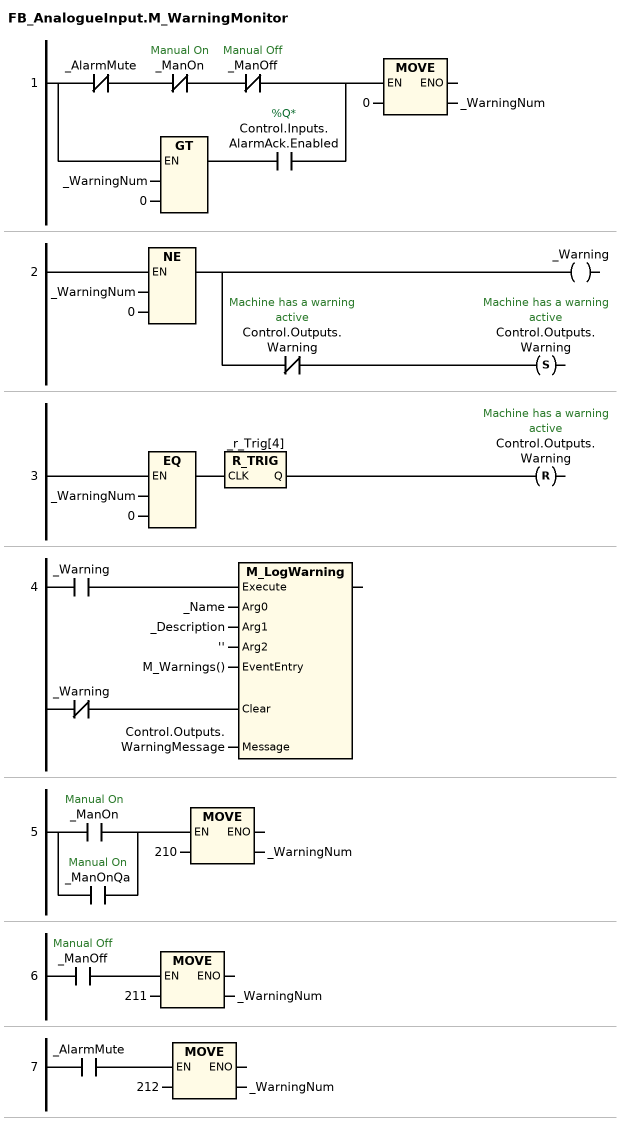
// NETWORK 1
//   _ManOn: Manual On
//   _ManOff: Manual Off
//   Control.Inputs.AlarmAck.Enabled: AT %Q*
IF NOT _AlarmMute AND NOT _ManOn AND NOT _ManOff OR _WarningNum > 0 AND Control.Inputs.AlarmAck.Enabled THEN
    _WarningNum := 0;
END_IF

// NETWORK 2
//   Control.Outputs.Warning: Machine has a warning active
_w1 := _WarningNum <> 0;
_Warning := _w1;
Control.Outputs.Warning S= _w1 AND NOT Control.Outputs.Warning;

// NETWORK 3
//   Control.Outputs.Warning: Machine has a warning active
_r_Trig[4](CLK := _WarningNum = 0); // R_TRIG
Control.Outputs.Warning R= _r_Trig[4].Q;

// NETWORK 4
M_LogWarning(Execute := _Warning, Arg0 := _Name, Arg1 := _Description, Arg2 := '', EventEntry := M_Warnings(), Clear := NOT _Warning, Message := Control.Outputs.WarningMessage);

// NETWORK 5
//   _ManOn: Manual On
//   _ManOnQa: Manual On
IF _ManOn OR _ManOnQa THEN _WarningNum := 210; END_IF

// NETWORK 6
//   _ManOff: Manual Off
IF _ManOff THEN _WarningNum := 211; END_IF

// NETWORK 7
IF _AlarmMute THEN _WarningNum := 212; END_IF
END_METHOD

METHOD PRIVATE M_Warnings : TcEventEntry
VAR_INPUT
END_VAR
CASE _WarningNum OF
	210: M_Warnings:= TC_Events.TcAnalogueInput.W_210;//Manual ON Enabled
	211: M_Warnings:= TC_Events.TcAnalogueInput.W_211;//Manual OFF Enabled			
	212: M_Warnings:= TC_Events.TcAnalogueInput.W_212;//Alarm Mute Active						
ELSE
	M_Warnings:=  TC_Events.TcAnalogueInput.W_Undefined;
END_CASE
END_METHOD

{attribute 'monitoring' := 'variable'}
PROPERTY PUBLIC ManOff : Bool
GET
ManOff := _ManOff;
END_GET
SET
_ManOff := ManOff;
END_SET
END_PROPERTY

{attribute 'monitoring' := 'variable'}
PROPERTY PUBLIC ManOn : Bool
GET
ManOn := _ManOn;
END_GET
SET
_ManOn := ManOn;
END_SET
END_PROPERTY

{attribute 'monitoring' := 'variable'}
PROPERTY PUBLIC ManOnQa : Bool
GET
ManOnQa := _ManOnQa;
END_GET
SET
_ManOnQa := ManOnQa;
END_SET
END_PROPERTY

{attribute 'monitoring' := 'variable'}
PROPERTY PUBLIC ManQa : REAL
GET
ManQa := _ManQa;
END_GET
SET
_ManQa := ManQa;
END_SET
END_PROPERTY

{attribute 'monitoring' := 'variable'}
PROPERTY PUBLIC Name : String[15]
GET
Name := _Name;
END_GET
SET
_Name := Name;
END_SET
END_PROPERTY

{attribute 'monitoring' := 'variable'}
PROPERTY PUBLIC RisingEdge : Bool
GET
RisingEdge := _RisingEdge;
END_GET
END_PROPERTY

{attribute 'monitoring' := 'variable'}
PROPERTY PUBLIC SimInput : Bool
SET
_SimInput := SimInput;
END_SET
END_PROPERTY

{attribute 'monitoring' := 'variable'}
PROPERTY PUBLIC SimInput2 : Bool
SET
_SimInput2 := SimInput2;
END_SET
END_PROPERTY

{attribute 'monitoring' := 'variable'}
PROPERTY PUBLIC SimInputQa : REAL
GET
SimInputQa := _SimInputQa;
END_GET
SET
_SimInputQa := SimInputQa;
END_SET
END_PROPERTY

{attribute 'monitoring' := 'variable'}
PROPERTY PUBLIC StandbyReset : Bool
GET
StandbyReset := _ForceOff;
END_GET
SET
_ForceOff := StandbyReset;
END_SET
END_PROPERTY

{attribute 'monitoring' := 'variable'}
PROPERTY PUBLIC Value_Q : BOOL
GET
Value_Q := _Value_Q;
END_GET
SET
_Value_Q := Value_Q;
END_SET
END_PROPERTY

{attribute 'monitoring' := 'variable'}
PROPERTY PUBLIC Value_Qa : REAL
GET
Value_Qa := _Value_Qa;
END_GET
SET
_Value_Qa := Value_Qa;
END_SET
END_PROPERTY

{attribute 'monitoring' := 'variable'}
PROPERTY PUBLIC Warning : Bool
GET
Warning := _Warning;
END_GET
END_PROPERTY

END_FUNCTION_BLOCK

// Objects/FB_EventLogger_V4_02/FB_EventLogger
FUNCTION_BLOCK FB_EventLogger
VAR
END_VAR

METHOD PROTECTED M_LogAlarm : BOOL;
VAR_INPUT
	Execute				: BOOL;					//Trigger Event
	Arg0				: STRING;				//Event Argument {0}
	Arg1				: STRING;				//Event Argument {1}
	Arg2				: STRING;				//Event Argument {2}
	EventEntry			: TcEventEntry;			//Alarm Event Entry
	Clear				: BOOL;					// Set Event to Not Raised
END_VAR
VAR_INST
	{attribute 'tc_no_symbol'}
	_fb_Alarm			: FB_TcAlarm;			//Event Logger Function Block
	{attribute 'tc_no_symbol'}
	_TcEventState		: USINT;     			//Event Logger State
	{attribute 'tc_no_symbol'}
	_TcEventError		: BOOL;      			//Event Text Request Error
	{attribute 'tc_no_symbol'}
	_TcEventText		: STRING;      			//Event Text
	{attribute 'tc_no_symbol'}
	_TcEventTrig		: R_TRIG;    			//Event Trigger
	{attribute 'tc_no_symbol'}
	_TcClearEventTrig	: R_TRIG;    			//Clear Event Trigger
	{attribute 'tc_no_symbol'}
	_TextRequest		: BOOL;					//Text Request Successful
END_VAR
VAR_IN_OUT
	Message				: STRING;				//Active Alarm Message
END_VAR
_TcEventTrig(CLK:=Execute);
CASE _TcEventState OF
0://Wait for Alarm
	IF _TcEventTrig.Q  AND EventEntry.nEventId > 0 THEN
		_TcEventState := 1;
	END_IF
1://Queue Alarm Event
	_fb_Alarm.CreateEx(stEventEntry:= EventEntry, bWithConfirmation:= TRUE, ipSourceInfo:= 0);
	_TcEventState := 2;
2://Set Arguments
	_fb_Alarm.ipArguments.Clear();
	IF (Arg1 = '' AND Arg0 <> '') THEN
		_fb_Alarm.ipArguments.AddString(Arg0);
	ELSIF (Arg2 = '' AND Arg1 <> '') THEN
		_fb_Alarm.ipArguments.AddString(Arg0).AddString(Arg1);
	ELSIF (Arg0 <> '' AND Arg1 <> '' AND Arg2 <> '') THEN
		_fb_Alarm.ipArguments.AddString(Arg0).AddString(Arg1).AddString(Arg2);
	END_IF
	_TcEventState := 3;
3://Raise Alarm
	_fb_Alarm.Raise(0);
	_TcEventError := FALSE;
	_TcEventState := 4;
4://Request Event Text
	_TextRequest := _fb_Alarm.RequestEventText(nLangId:= 1033, sResult:= _TcEventText, nResultSize:= SIZEOF(_TcEventText), bError=> _TcEventError, hrErrorCode=>);
	IF _TextRequest OR _TcEventError THEN
		IF _TcEventError THEN _TcEventText := 'Error Requesting Event Text'; END_IF
		_TcEventState := 5;
	END_IF
5://Return Active Alarm Message
	Message := CONCAT('[',CONCAT(UDINT_TO_STRING(_fb_Alarm.nEventId),CONCAT('] - ', _TcEventText)));	
	_TcEventState := 0;
END_CASE

// Clears Alarm
_TcClearEventTrig(CLK:= Clear AND NOT Execute);
IF _TcClearEventTrig.Q THEN
	_fb_Alarm.Clear(nTimeStamp:= 0, bResetConfirmation:= FALSE);
	_fb_Alarm.Confirm(nTimeStamp:= 0);
END_IF

//Alarm Logging Not Busy
M_LogAlarm := _TcEventState = 0;
END_METHOD

METHOD PROTECTED M_LogAlert : BOOL;
VAR_INPUT
	Execute				: BOOL;					//Trigger Event
	Arg0				: STRING;				//Event Argument {0}
	Arg1				: STRING;				//Event Argument {1}
	Arg2				: STRING;				//Event Argument {2}
	EventEntry			: TcEventEntry;			//Alert Event Entry 
END_VAR
VAR_INST
	{attribute 'tc_no_symbol'}
	_fb_Alert			: FB_TcMessage;			//Event Logger Function Block
	{attribute 'tc_no_symbol'}
	_TcEventState		: USINT;     			//Event Logger State
	{attribute 'tc_no_symbol'}
	_TcEventError		: BOOL;      			//Event Text Request Error
	{attribute 'tc_no_symbol'}
	_TcEventText		: STRING;      			//Event Text
	{attribute 'tc_no_symbol'}
	_TcEventTrig		: R_TRIG;    			//Event Trigger
	{attribute 'tc_no_symbol'}
	_TextRequest		: BOOL;					//Text Request Successful
END_VAR
VAR_IN_OUT
	Message				: STRING;				//Active Alert Message
END_VAR
_TcEventTrig(CLK:=Execute);
CASE _TcEventState OF
0://Wait for Alert
	IF _TcEventTrig.Q AND EventEntry.nEventId > 0 THEN
		_TcEventState := 1;
	END_IF
1://Queue Alert Event
	_fb_Alert.CreateEx(stEventEntry:= EventEntry, ipSourceInfo:= 0);
	_TcEventState := 2;
2://Set Arguments
	_fb_Alert.ipArguments.Clear();
	IF (Arg1 = '' AND Arg0 <> '') THEN
		_fb_Alert.ipArguments.AddString(Arg0);
	ELSIF (Arg2 = '' AND Arg1 <> '') THEN
		_fb_Alert.ipArguments.AddString(Arg0).AddString(Arg1);
	ELSIF (Arg0 <> '' AND Arg1 <> '' AND Arg2 <> '') THEN
		_fb_Alert.ipArguments.AddString(Arg0).AddString(Arg1).AddString(Arg2);
	END_IF
	_TcEventState := 3;
3://Raise Alert
	_fb_Alert.Send(0);
	_TcEventState := 4;
4://Request Event Text
	_TcEventError := FALSE;
	_TextRequest:= _fb_Alert.RequestEventText(nLangId:= 1033, sResult:= _TcEventText, nResultSize:= SIZEOF(_TcEventText), bError=> _TcEventError, hrErrorCode=> ) ;
	IF _TextRequest OR _TcEventError THEN
		IF _TcEventError THEN Message := 'Error Requesting Event Text'; END_IF
		_TcEventState := 5;
	END_IF
5://Return Active Alert Message
	Message := CONCAT('[',CONCAT(UDINT_TO_STRING(_fb_Alert.nEventId),CONCAT('] - ', _TcEventText)));	
	_TcEventState := 0;
END_CASE

//Alert Logging Not Busy
M_LogAlert := _TcEventState = 0;
END_METHOD

METHOD PROTECTED M_LogMessage : BOOL;
VAR_INPUT
	Execute				: BOOL;					//Trigger Event
	Arg0				: STRING;				//Event Argument {0}
	Arg1				: STRING;				//Event Argument {1}
	Arg2				: STRING;				//Event Argument {2}
	EventEntry			: TcEventEntry;			//Alarm Event Entry 
END_VAR
VAR_INST
	{attribute 'tc_no_symbol'}
	_fb_Message			: FB_TcMessage;			//Event Logger Function Block
	{attribute 'tc_no_symbol'}
	_TcEventState		: USINT;     			//Event Logger State
	{attribute 'tc_no_symbol'}
	_TcEventTrig		: R_TRIG;    			//Event Trigger
END_VAR
_TcEventTrig(CLK:=Execute);
CASE _TcEventState OF
0://Wait for Message
	IF _TcEventTrig.Q AND EventEntry.nEventId > 0 THEN
		_TcEventState := 1;
	END_IF
1://Queue Message Event
	_fb_Message.CreateEx(EventEntry, 0);
	_TcEventState := 2;
2://Set Arguments
	_fb_Message.ipArguments.Clear();
	IF (Arg1 = '' AND Arg0 <> '') THEN
		_fb_Message.ipArguments.AddString(Arg0);
	ELSIF (Arg2 = '' AND Arg1 <> '') THEN
		_fb_Message.ipArguments.AddString(Arg0).AddString(Arg1);
	ELSIF (Arg0 <> '' AND Arg1 <> '' AND Arg2 <> '') THEN
		_fb_Message.ipArguments.AddString(Arg0).AddString(Arg1).AddString(Arg2);
	END_IF
	_TcEventState := 3;
3://Raise Warning
	_fb_Message.Send(0);
	_TcEventState := 0;
END_CASE

//Message Logging Not Busy
M_LogMessage := _TcEventState = 0;
END_METHOD

METHOD PROTECTED M_LogWarning : BOOL;
VAR_INPUT
	Execute				: BOOL;					//Trigger Event
	Arg0				: STRING;				//Event Argument {0}
	Arg1				: STRING;				//Event Argument {1}
	Arg2				: STRING;				//Event Argument {2}
	EventEntry			: TcEventEntry;			//Alarm Event Entry 
	Clear				: BOOL;					//Set Event to Not Raised
END_VAR
VAR_INST
	{attribute 'tc_no_symbol'}
	_fb_Warning			: FB_TcAlarm;			//Event Logger Function Block
	{attribute 'tc_no_symbol'}
	_TcEventState		: USINT;     			//Event Logger State
	{attribute 'tc_no_symbol'}
	_TcEventError		: BOOL;      			//Event Text Request Error
	{attribute 'tc_no_symbol'}
	_TcEventText		: STRING;      			//Event Text
	{attribute 'tc_no_symbol'}
	_TcEventTrig		: R_TRIG;    			//Event Trigger
	{attribute 'tc_no_symbol'}
	_TcClearEventTrig	: R_TRIG;    			//Clear Event Trigger
	{attribute 'tc_no_symbol'}
	_TextRequest		: BOOL;					//Text Request Successful
END_VAR
VAR_IN_OUT
	Message				: STRING;				//Active Warning Message
END_VAR
_TcEventTrig(CLK:=Execute);
CASE _TcEventState OF
0://Wait for Warning
	IF _TcEventTrig.Q AND EventEntry.nEventId > 0 THEN
		_TcEventState := 1;
	END_IF
1://Queue Warning Event
	_fb_Warning.CreateEx(stEventEntry:= EventEntry,bWithConfirmation:= TRUE, ipSourceInfo:= 0);
	_TcEventState := 2;
2://Set Arguments
	_fb_Warning.ipArguments.Clear();
	IF (Arg1 = '' AND Arg0 <> '') THEN
		_fb_Warning.ipArguments.AddString(Arg0);
	ELSIF (Arg2 = '' AND Arg1 <> '') THEN
		_fb_Warning.ipArguments.AddString(Arg0).AddString(Arg1);
	ELSIF (Arg0 <> '' AND Arg1 <> '' AND Arg2 <> '') THEN
		_fb_Warning.ipArguments.AddString(Arg0).AddString(Arg1).AddString(Arg2);
	END_IF
	_TcEventState := 3;
3://Raise Warning
	_fb_Warning.Raise(0);
	_TcEventState := 4;
4://Request Event Text
	_TcEventError := FALSE;
	_TextRequest := _fb_Warning.RequestEventText(nLangId:= 1033, sResult:= _TcEventText, nResultSize:= SIZEOF(_TcEventText), bError=> _TcEventError, hrErrorCode=> ) ;
	IF _TextRequest OR _TcEventError THEN
		IF _TcEventError THEN Message := 'Error Requesting Event Text'; END_IF
		_TcEventState := 5;
	END_IF
5://Return Active Warning Message
	Message := CONCAT('[',CONCAT(UDINT_TO_STRING(_fb_Warning.nEventId),CONCAT('] - ', _TcEventText)));
	_TcEventState := 0;
END_CASE
	
// Clears Alarm
_TcClearEventTrig(CLK:=Clear AND NOT Execute);
IF _TcClearEventTrig.Q THEN
	_fb_Warning.Clear(nTimeStamp:= 0, bResetConfirmation:= FALSE);
	_fb_Warning.Confirm(nTimeStamp:= 0);
END_IF

//Warning Logging Not Busy
M_LogWarning := _TcEventState = 0;
END_METHOD

END_FUNCTION_BLOCK

// Objects/FB_AnalogueOutput_V4_01/FB_AnalogueOutput
FUNCTION_BLOCK FINAL FB_AnalogueOutput EXTENDS FB_EventLogger
VAR_IN_OUT
	Control					: ST_System;
END_VAR
VAR
	_Input					: UINT;					//Raw Input 1 - Analogue
	_Input2					: BOOL;					//Raw Input 2 - Digital
	_ManOnQa				: BOOL;					//Manual On Analogue Input
	_ManQa					: REAL;					//Manual Analogue Input
	_ManOn					: BOOL;					//Manual On
	_ManOff					: BOOL;					//Manual Off
	_ForceOn				: BOOL;					//Force On
	_ForceOff				: BOOL;					//Force Off
	_Fault					: BOOL;					//Fault
	_SimInput				: BOOL;  				//Simulates Analogue Input
	_SimInput2				: BOOL;					//Simulates Digital Input
	_SimInputQa				: REAL;					//Value of Simulated Analogue Input
	_Value_Q	AT %Q*		: BOOL;					//Value of Input - Digital
	_Value_Qa	AT %Q*		: INT;					//Value of Input - Analogue
	_FallingEdge			: BOOL;					//Falling Edge of Value Signal
	_RisingEdge				: BOOL;					//Raising Edge of Value Signal
	_DebounceOn_ET			: REAL;					//Debounce On Elapsed Time
	_DebounceOff_ET			: REAL;					//Debounce Off Elapsed Time
	_FaultTimer_ET			: REAL;					//Fault timer elapsed
	_HighAlarmLimit			: BOOL;					//Input Value is approaching the maximum operating limit.
	_LowAlarmLimit			: BOOL;					//Input Value is approaching the minimum operating limit.
	_HighHighAlarmLimit		: BOOL;					//Input Value is above  the maximum operating limit
	_LowLowAlarmLimit		: BOOL;					//Input Value is below the minimum operating limit.
	_Alarm					: BOOL;					//Device Alarm
	_Warning				: BOOL;					//Device Warning
	_AlarmNum				: DINT;					//Device Alarm Number
	_WarningNum				: DINT;					//Device Warning Number
	_riseEdge				: R_TRIG;				//Rising Edge Value Trigger
	_fallEdge				: F_TRIG;				//Falling Edge Value Trigger
	_ConfInput				: BOOL;					//Confirgured Input
	_DebounceOn_DN			: BOOL;					//Debounce On Timer is Done
	_DebounceOff_DN			: BOOL;					//Debounce Off Timer is Done
	_R_Trig					: ARRAY[0..9] OF R_TRIG;//Private Rising Edge Triggers
END_VAR
VAR PERSISTENT
	_Name					: STRING[15];			//Name for HMI
	_Description			: STRING[40];			//Description for HMI
	_AlarmMute				: BOOL;					//Alarm Mute
	_TypeConfig				: E_AOutputTypeConfig;	//Type congifuration
	_DebounceOn_PT			: REAL;					//Debounce on timer preset time
	_DebounceOff_PT			: REAL;					//Debounce off timer preset time
	_FaultTimer_PT			: REAL;					//Fault timer preset time
	_InputLimitHigh			: REAL;					//HighHigh limit of Raw Input 1
	_InputLimitLow			: REAL;					//Low limit of Raw Input 1
	_InputLimitHighHigh		: REAL;					//HighHigh limit of Raw Input 1
	_InputLimitLowLow		: REAL;					//LowLow limit of Raw Input 1
	_Scale_Qa				: REAL;					//Scale Factor
	_Subtract_Qa			: REAL;					//Subtract a constant from the output
	_Add_Qa					: REAL;					//Add a constant to the output
END_VAR

M_TypeConfig();
M_AlarmMonitor();
M_WarningMonitor();
M_UnlatchManuals();
M_Output();

//Debounce On Timer
IF _ConfInput = TRUE AND NOT _ForceOff AND NOT _ManOff THEN
	_DebounceOn_ET := _DebounceOn_ET + Control.SystemTime.ScanTime;
	_debounceOn_DN := _DebounceOn_ET > _DebounceOn_PT;
ELSE
	_debounceOn_DN := FALSE;
END_IF
IF _debounceOn_DN OR _ForceOn OR _ManOn THEN
	_Value_Q := TRUE;
	_DebounceOff_ET := 0;
END_IF

//Debounce Off Timer
IF _ConfInput = FALSE AND NOT _ForceOn AND NOT _ManOn THEN
	_DebounceOff_ET := _DebounceOff_ET + Control.SystemTime.ScanTime;
	_debounceOff_DN := _DebounceOff_ET > _DebounceOff_PT;
ELSE
	_debounceOff_DN := FALSE;
END_IF
IF _debounceOff_DN OR _ForceOff OR _ManOff THEN
	_Value_Q:= FALSE;
	_DebounceOn_ET := 0;
END_IF

//Rising Edge Trigger 
_riseEdge(CLK := _Value_Q);
_RisingEdge := _riseEdge.Q;

//Falling Edge Trigger
_fallEdge(CLK := _Value_Q);
_FallingEdge := _fallEdge.Q;

{attribute 'monitoring' := 'variable'}
PROPERTY PUBLIC Alarm : Bool
GET
Alarm := _Alarm;
END_GET
END_PROPERTY

{attribute 'monitoring' := 'variable'}
PROPERTY PUBLIC AlarmMute : BOOL
SET
AlarmMute := _AlarmMute;
END_SET
END_PROPERTY

{attribute 'monitoring' := 'variable'}
PROPERTY PUBLIC DebounceOff_ET : real
GET
DebounceOff_ET := _DebounceOff_ET;
END_GET
END_PROPERTY

{attribute 'monitoring' := 'variable'}
PROPERTY PUBLIC DebounceOff_PT : real
GET
DebounceOff_PT := _DebounceOff_PT;
END_GET
SET
_DebounceOff_PT := DebounceOff_PT;
END_SET
END_PROPERTY

{attribute 'monitoring' := 'variable'}
PROPERTY PUBLIC DebounceOn_ET : real
GET
DebounceOn_ET := _DebounceOn_ET;
END_GET
END_PROPERTY

{attribute 'monitoring' := 'variable'}
PROPERTY PUBLIC DebounceOn_PT : real
GET
DebounceOn_PT := _DebounceOn_PT;
END_GET
SET
_DebounceOn_PT := DebounceOn_PT;
END_SET
END_PROPERTY

{attribute 'monitoring' := 'variable'}
PROPERTY PUBLIC Description : String[40]
GET
Description := _Description;
END_GET
SET
_Description := Description;
END_SET
END_PROPERTY

{attribute 'monitoring' := 'variable'}
PROPERTY PUBLIC FallingEdge : Bool
GET
FallingEdge := _FallingEdge;
END_GET
END_PROPERTY

{attribute 'monitoring' := 'variable'}
PROPERTY PUBLIC Fault : Bool
SET
_Fault := Fault;
END_SET
END_PROPERTY

{attribute 'monitoring' := 'variable'}
PROPERTY PUBLIC FaultTimer_ET : real
GET
FaultTimer_ET := _FaultTimer_ET;
END_GET
END_PROPERTY

{attribute 'monitoring' := 'variable'}
PROPERTY PUBLIC FaultTimer_PT : real
GET
FaultTimer_PT := _FaultTimer_PT;
END_GET
SET
_FaultTimer_PT := FaultTimer_PT;
END_SET
END_PROPERTY

{attribute 'monitoring' := 'variable'}
PROPERTY PUBLIC ForceOn : Bool
GET
ForceOn := _ForceOn;
END_GET
SET
_ForceOn := ForceOn;
END_SET
END_PROPERTY

{attribute 'monitoring' := 'variable'}
PROPERTY PUBLIC Input : UINT
GET
Input := _Input;
END_GET
SET
PUBLIC 
VAR
END_VAR
_Input := Input;
END_SET
END_PROPERTY

{attribute 'monitoring' := 'variable'}
PROPERTY PUBLIC Input2 : Bool
GET
Input2 := _Input2;
END_GET
END_PROPERTY

METHOD PRIVATE M_AlarmMonitor
VAR_INPUT
END_VAR
VAR_INST
END_VAR
VAR_INST // added by the converter: edge detectors and wires of the graphical bodies
    _w1, _w2, _w3, _w4, _w5 : BOOL;
END_VAR
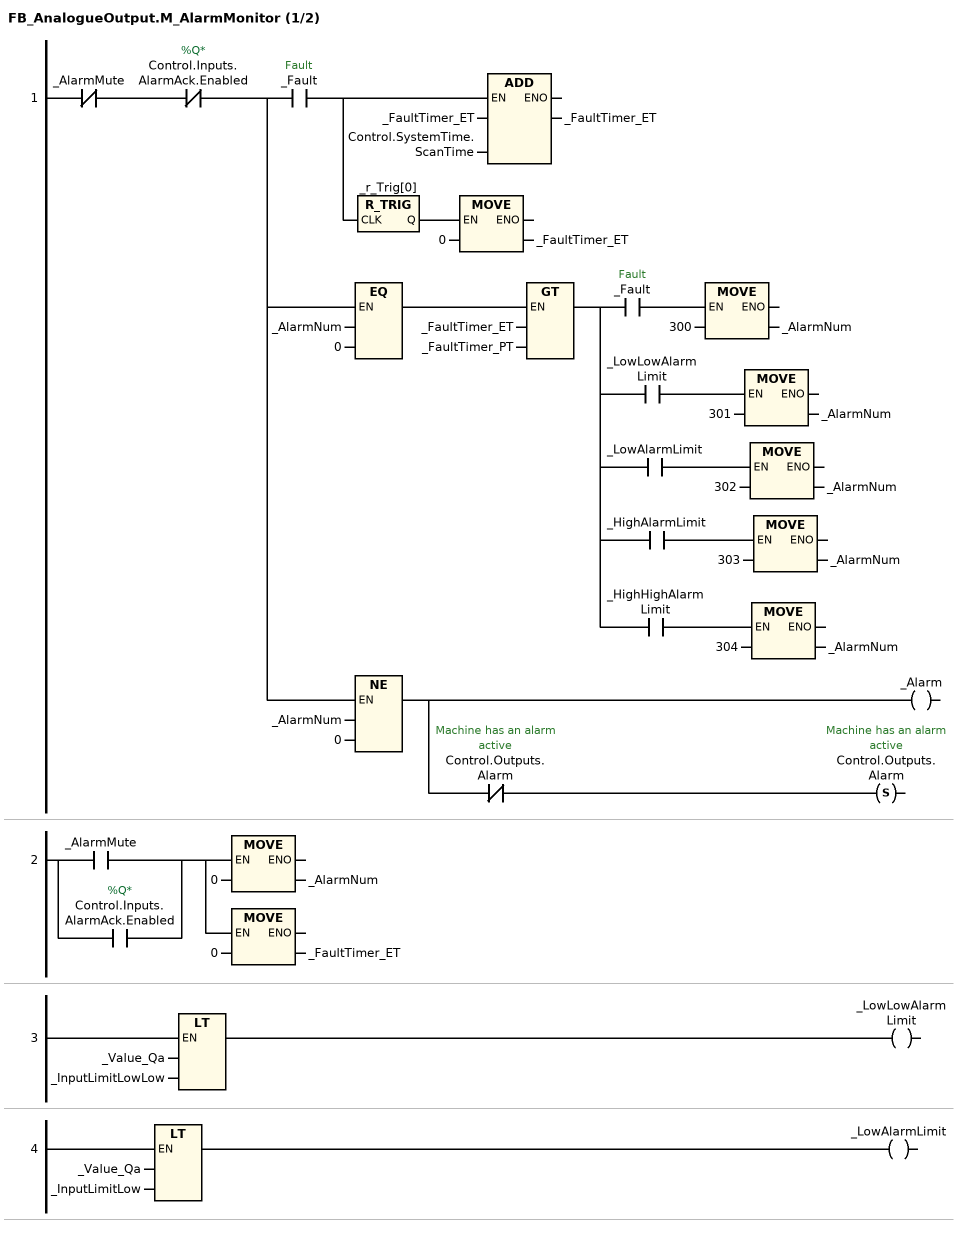
// NETWORK 1
//   Control.Inputs.AlarmAck.Enabled: AT %Q*
//   _Fault: Fault
//   _FaultTimer_ET: Fault timer elapsed
//   Control.SystemTime.ScanTime: Last scan time (Seconds)
//   _FaultTimer_PT: Fault timer preset time
//   Control.Outputs.Alarm: Machine has an alarm active
_w1 := NOT _AlarmMute AND NOT Control.Inputs.AlarmAck.Enabled;
_w2 := _w1 AND _Fault;
IF _w2 THEN _FaultTimer_ET := _FaultTimer_ET + Control.SystemTime.ScanTime; END_IF
_r_Trig[0](CLK := _w2); // R_TRIG
IF _r_Trig[0].Q THEN _FaultTimer_ET := 0; END_IF
_w3 := _w1 AND _AlarmNum = 0 AND _FaultTimer_ET > _FaultTimer_PT;
IF _w3 AND _Fault THEN _AlarmNum := 300; END_IF
IF _w3 AND _LowLowAlarmLimit THEN _AlarmNum := 301; END_IF
IF _w3 AND _LowAlarmLimit THEN _AlarmNum := 302; END_IF
IF _w3 AND _HighAlarmLimit THEN _AlarmNum := 303; END_IF
IF _w3 AND _HighHighAlarmLimit THEN _AlarmNum := 304; END_IF
_w4 := _w1 AND _AlarmNum <> 0;
_Alarm := _w4;
Control.Outputs.Alarm S= _w4 AND NOT Control.Outputs.Alarm;

// NETWORK 2
//   Control.Inputs.AlarmAck.Enabled: AT %Q*
//   _FaultTimer_ET: Fault timer elapsed
_w5 := _AlarmMute OR Control.Inputs.AlarmAck.Enabled;
IF _w5 THEN _AlarmNum := 0; END_IF
IF _w5 THEN _FaultTimer_ET := 0; END_IF

// NETWORK 3
_LowLowAlarmLimit := _Value_Qa < _InputLimitLowLow;

// NETWORK 4
_LowAlarmLimit := _Value_Qa < _InputLimitLow;

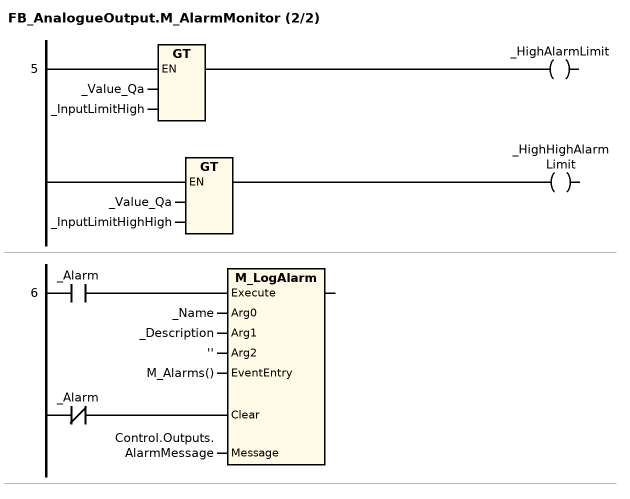
// NETWORK 5
_HighAlarmLimit := _Value_Qa > _InputLimitHigh;
_HighHighAlarmLimit := _Value_Qa > _InputLimitHighHigh;

// NETWORK 6
M_LogAlarm(Execute := _Alarm, Arg0 := _Name, Arg1 := _Description, Arg2 := '', EventEntry := M_Alarms(), Clear := NOT _Alarm, Message := Control.Outputs.AlarmMessage);
END_METHOD

METHOD PRIVATE M_Alarms : TcEventEntry
VAR_INPUT
END_VAR
CASE _AlarmNum OF
	301: M_Alarms:= TC_Events.TcAnalogueOutput.A_301;//Low Low Limit Alarm	
	302: M_Alarms:= TC_Events.TcAnalogueOutput.A_302;//Low Limit Alarm			
	303: M_Alarms:= TC_Events.TcAnalogueOutput.A_303;//High Limit Alarm
	304: M_Alarms:= TC_Events.TcAnalogueOutput.A_304;//High High Limit Alarm							
ELSE
	M_Alarms:= TC_Events.TcAnalogueOutput.A_Undefined;
END_CASE
END_METHOD

METHOD PRIVATE M_Output
VAR_INPUT
END_VAR
VAR_INST
END_VAR
IF _ManOnQa THEN
	IF _Scale_Qa <> 0 THEN
		_Value_Qa :=REAL_TO_INT(_ManQa * _Scale_Qa);
	ELSE
		_Value_Qa :=REAL_TO_INT(_ManQa);
	END_IF	
	
ELSIF _SimInput THEN
	IF _Scale_Qa <> 0 THEN
		_Value_Qa :=REAL_TO_INT(_SimInputQa * _Scale_Qa);
	ELSE
		_Value_Qa :=REAL_TO_INT(_SimInputQa);
	END_IF
	
ELSE
	IF _Scale_Qa <> 0 THEN
		_Value_Qa :=REAL_TO_INT((_Input + _Add_Qa - _Subtract_Qa) * _Scale_Qa);
	ELSE
		_Value_Qa :=REAL_TO_INT( _Input + _Add_Qa - _Subtract_Qa);
	END_IF	
END_IF
END_METHOD

METHOD PRIVATE M_TypeConfig
VAR_INPUT
END_VAR
VAR_INST
END_VAR
CASE _TypeConfig OF
	eAOutputType_PLC_NO, eAOutputType_SAFE_NO : 
		IF _Input2 OR _SimInput2 THEN
			_ConfInput := TRUE;
		ELSE
			_ConfInput := FALSE;
		END_IF
	eAOutputType_PLC_NC, eAOutputType_SAFE_NC : 
		IF NOT _Input2 OR _SimInput2 THEN
			_ConfInput := TRUE;
		ELSE
			_ConfInput := FALSE;
		END_IF
END_CASE
END_METHOD

METHOD PRIVATE M_UnlatchManuals
VAR_INPUT
END_VAR
VAR_INST
END_VAR
VAR_INST // added by the converter: edge detectors and wires of the graphical bodies
    _rt1, _rt2, _rt3 : R_TRIG;
END_VAR
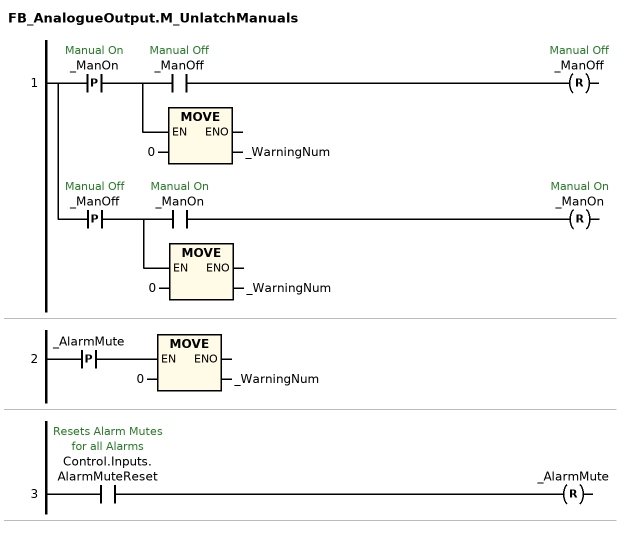
// NETWORK 1
//   _ManOn: Manual On
//   _ManOff: Manual Off
_rt1(CLK := _ManOn);
_ManOff R= _rt1.Q AND _ManOff;
IF _rt1.Q THEN _WarningNum := 0; END_IF
_rt2(CLK := _ManOff);
_ManOn R= _rt2.Q AND _ManOn;
IF _rt2.Q THEN _WarningNum := 0; END_IF

// NETWORK 2
_rt3(CLK := _AlarmMute);
IF _rt3.Q THEN _WarningNum := 0; END_IF

// NETWORK 3
//   Control.Inputs.AlarmMuteReset: Resets Alarm Mutes for all Alarms
_AlarmMute R= Control.Inputs.AlarmMuteReset;
END_METHOD

METHOD PRIVATE M_WarningMonitor
VAR_INPUT
END_VAR
VAR_INST
END_VAR
VAR_INST // added by the converter: edge detectors and wires of the graphical bodies
    _w1 : BOOL;
END_VAR
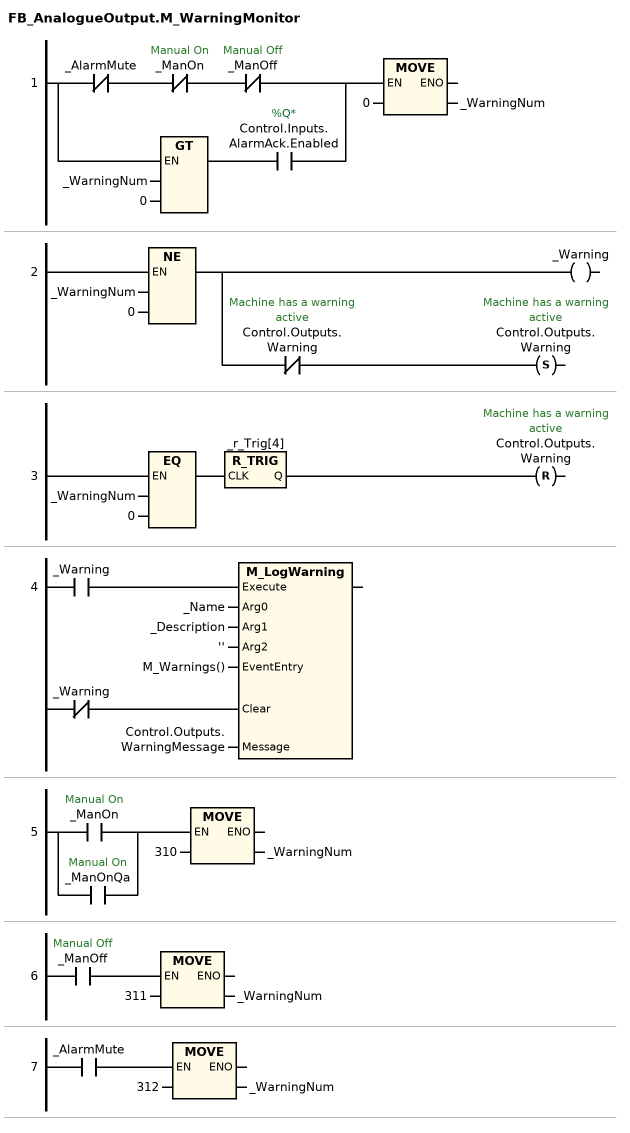
// NETWORK 1
//   _ManOn: Manual On
//   _ManOff: Manual Off
//   Control.Inputs.AlarmAck.Enabled: AT %Q*
IF NOT _AlarmMute AND NOT _ManOn AND NOT _ManOff OR _WarningNum > 0 AND Control.Inputs.AlarmAck.Enabled THEN
    _WarningNum := 0;
END_IF

// NETWORK 2
//   Control.Outputs.Warning: Machine has a warning active
_w1 := _WarningNum <> 0;
_Warning := _w1;
Control.Outputs.Warning S= _w1 AND NOT Control.Outputs.Warning;

// NETWORK 3
//   Control.Outputs.Warning: Machine has a warning active
_r_Trig[4](CLK := _WarningNum = 0); // R_TRIG
Control.Outputs.Warning R= _r_Trig[4].Q;

// NETWORK 4
M_LogWarning(Execute := _Warning, Arg0 := _Name, Arg1 := _Description, Arg2 := '', EventEntry := M_Warnings(), Clear := NOT _Warning, Message := Control.Outputs.WarningMessage);

// NETWORK 5
//   _ManOn: Manual On
//   _ManOnQa: Manual On
IF _ManOn OR _ManOnQa THEN _WarningNum := 310; END_IF

// NETWORK 6
//   _ManOff: Manual Off
IF _ManOff THEN _WarningNum := 311; END_IF

// NETWORK 7
IF _AlarmMute THEN _WarningNum := 312; END_IF
END_METHOD

METHOD PRIVATE M_Warnings : TcEventEntry
VAR_INPUT
END_VAR
CASE _WarningNum OF
	310: M_Warnings:= TC_Events.TcAnalogueOutput.W_310;//Manual ON Enabled	
	311: M_Warnings:= TC_Events.TcAnalogueOutput.W_311;//Manual OFF Enabled			
	312: M_Warnings:= TC_Events.TcAnalogueOutput.W_312;//Alarm Mute Active					
ELSE
	M_Warnings:=  TC_Events.TcAnalogueOutput.W_Undefined;
END_CASE
END_METHOD

{attribute 'monitoring' := 'variable'}
PROPERTY PUBLIC ManOff : Bool
GET
ManOff := _ManOff;
END_GET
SET
_ManOff := ManOff;
END_SET
END_PROPERTY

{attribute 'monitoring' := 'variable'}
PROPERTY PUBLIC ManOn : Bool
GET
ManOn := _ManOn;
END_GET
SET
_ManOn := ManOn;
END_SET
END_PROPERTY

{attribute 'monitoring' := 'variable'}
PROPERTY PUBLIC ManOnQa : Bool
GET
ManOnQa := _ManOnQa;
END_GET
SET
_ManOnQa := ManOnQa;
END_SET
END_PROPERTY

{attribute 'monitoring' := 'variable'}
PROPERTY PUBLIC ManQa : REAL
GET
ManQa := _ManQa;
END_GET
SET
_ManQa := ManQa;
END_SET
END_PROPERTY

{attribute 'monitoring' := 'variable'}
PROPERTY PUBLIC Name : String[15]
GET
Name := _Name;
END_GET
SET
_Name := Name;
END_SET
END_PROPERTY

{attribute 'monitoring' := 'variable'}
PROPERTY PUBLIC RisingEdge : Bool
GET
RisingEdge := _RisingEdge;
END_GET
END_PROPERTY

{attribute 'monitoring' := 'variable'}
PROPERTY PUBLIC SimInput : Bool
SET
_SimInput := SimInput;
END_SET
END_PROPERTY

{attribute 'monitoring' := 'variable'}
PROPERTY PUBLIC SimInput2 : Bool
SET
_SimInput2 := SimInput2;
END_SET
END_PROPERTY

{attribute 'monitoring' := 'variable'}
PROPERTY PUBLIC SimInputQa : REAL
GET
SimInputQa := _SimInputQa;
END_GET
SET
_SimInputQa := SimInputQa;
END_SET
END_PROPERTY

{attribute 'monitoring' := 'variable'}
PROPERTY PUBLIC StandbyReset : Bool
GET
StandbyReset := _ForceOff;
END_GET
SET
_ForceOff := StandbyReset;
END_SET
END_PROPERTY

{attribute 'monitoring' := 'variable'}
PROPERTY PUBLIC Value_Q : BOOL
GET
Value_Q := _Value_Q;
END_GET
SET
_Value_Q := Value_Q;
END_SET
END_PROPERTY

{attribute 'monitoring' := 'variable'}
PROPERTY PUBLIC Value_Qa : INT
GET
Value_Qa := _Value_Qa;
END_GET
SET
_Value_Qa := Value_Qa;
END_SET
END_PROPERTY

{attribute 'monitoring' := 'variable'}
PROPERTY PUBLIC Warning : Bool
GET
Warning := _Warning;
END_GET
END_PROPERTY

END_FUNCTION_BLOCK

// Objects/FB_CNC_V1_01/FB_CNC
FUNCTION_BLOCK PUBLIC FB_CNC EXTENDS FB_EventLogger
VAR_INPUT
	CalibrationCam						: ARRAY[0..HLI_SYS_AX_MAXIDX] OF BOOL;
	LogAxisNo							: ARRAY[0..HLI_SYS_AX_MAXIDX] OF INT;// EtherCAT ID of Axis
	MaxChannelIdx						: INT := 0;	//Max index of channel that is used starting at 0, example: 1 -> totally 2 channels, maximum of 11 (12 channels) is allowed here *)
	Energize							: BOOL;// CNC Energised Flag
END_VAR
VAR_OUTPUT
	
END_VAR
VAR_IN_OUT	                			
	Control								: ST_System;
	Spindle								: ST_Spindle;						//Spindle interface	
END_VAR    
VAR 
	_AxisTorqueLimit					AT %Q* : ARRAY [0..4] OF UINT;								//Bipolar Torque Limit for axes (mapped from drive)
	_DrivePowerManagementStatusWords AT %I* :ARRAY [0..4] OF INT;									//Power management status to detect drives dropping power to ensure rehoming occurs.
	
	_Axis								: ARRAY[0..HLI_SYS_AX_MAXIDX] OF FB_CNCAxis;	//Axis data struct
	{attribute 'tc_no_symbol'}
	_Channel							: ARRAY[0..3] OF HLI3_CNCChannel;	//Channel data struct
	_MachineMode						: ARRAY[0..3] OF ST_MachineMode;	//Machine mode data struct
	_ManualMode							: ST_Selection;						//Manual Mode Selection
	_AutomaticMode						: ST_Selection;						//Automatic Mode Selection
	_MDIMode							: ST_Selection;						//MDI Mode Selection
	_HandwheelMode						: ST_Selection;						//Handwheel Mode Selection
	_StandbyMode						: ST_Selection;						//Standby Mode Selection
	_ReferenceMode						: ST_Selection;						//Reference Mode Selection
	_ManHome							: ST_Selection;						//Manual Home Selection
	_RetractTool						: ST_Selection;						//Retract tool from workpiece
	_SpindleWarmup						: ST_Selection;						//Warm up Spindle
	_AxisNames							: ARRAY[0..4] OF STRING;			//Individual Axis Names for HMI
	_AxisInManual						: ARRAY[0..4] OF BOOL;				//Axis in Manual Flag
	_SelectedChannel					: INT := 0;
	_SelectedAxis						: INT := 0;							//Axis Index Selected from HMI
	_SpindleVelocity					: UINT;								//Spindle Velocity Status
	_SpindleRev							: DINT;								//Spindle Revolution Command
	_AutoEn								: BOOL;								//Auto Enable
	_AutoHome							: BOOL;								//Command Home Drive Auto
	_AxisEnabled						: BOOL;								//All Axes are enabled
	_ManualModeJog						: BOOL;								//Manual Jog Mode
	_ManualModeInc						: BOOL;								//Manual Increment Mode
	_FeedOverride						: UINT := 100;
	_Fault								: BOOL;	     						//Device Fault
	_FaultTimer_ET						: REAL;								//Fault timer elapsed
	_Alarm								: BOOL;								//Device Alarm         
	_Warning							: BOOL;								//Device Warning   
	{attribute 'tc_no_symbol'}
	_ParkMDIString						: STRING;							//Parking MDI String   
	{attribute 'tc_no_symbol'}  
	_AlarmNum							: UDINT;							//Device Alarm Number  
	{attribute 'tc_no_symbol'}
	_WarningNum							: DINT;								//Device Warning Number
	{attribute 'tc_no_symbol'}
	_R_Trig								: ARRAY[0..19] OF R_TRIG;			//Private Rising Edge Triggers
	_HandwheelAxisIsSelected			: BOOL;								//True when axis selected on handwheel
	_Handwheel 							: ST_Handwheel; 					//Handwheel controller inputs
	_ProgramEnd							: ARRAY[0..3] OF BOOL;				//Program End
	_CurrentLine						: DINT;								//N function of currently running program (i.e. N60 -> 60)
	_CurrentNCProgram					: STRING;							//Program currently running in CNC kernal
	_NCProgramCode						: STRING(15000);					//Code of program for reloading into HMI text display\
END_VAR
VAR PERSISTENT                      	
	_Name								: STRING[15];						//Name for HMI
	_Description						: STRING[40];						//Description for HMI
	_AlarmMute							: BOOL;								//Alarm Mute
	_FaultTimer_PT						: REAL;								//Fault timer preset time	
	_Homed								: BOOL;								//Servo is Homed
	_Variables							: ARRAY [0..9] OF ST_Variable;				//Device Associated Varibles Array	
	_ToolData							: ARRAY [0..6] OF ST_CNC_TOOL_DATA_EXT;		//Data for tools
	_PositionOffset						: ARRAY[0..HLI_SYS_AX_MAXIDX] OF LREAL;		//Home position offsets for Axes
	_ParkPositions						: ARRAY[0..HLI_SYS_AX_MAXIDX] OF INT;		//Park positions for Axes
	_pVE_Chan0							: POINTER TO ST_VE_CHAN0;					//Channel 0 User defined Variables
	_Referencing						: E_CNC_HomingMethod; 						//Method to home
	_MeasurementOrder					: ARRAY[0..5] OF UINT :=[2,3,4,1,0];		//Measurement Axis Index Order i.e [2,3,4,1,0] Would be the same as G74 X5 Y4 Z1 C3 A2
	_MeasurementMDIString				: ARRAY[0..5] OF STRING := ['G100 X-10000$R$NM50$R$NM53$R$NG4 1$R$NM51$R$N#PUT AX [X] $R$NM52$R$N#CALL AX [X,11,0]$R$NM54$R$N',
																	'G100 Y-10000$R$NM50$R$NM53$R$NG4 1$R$NM51$R$N#PUT AX [Y] $R$NM52$R$N#CALL AX [Y,10,1]$R$NM54$R$N',
																	'G100 Z1000$R$NM50$R$NM53$R$NG4 1$R$NM51$R$N#PUT AX [Z] $R$NM52$R$N#CALL AX [Z,7,2]$R$NM54$R$N',
																	'G100 C-1000$R$NM50$R$NM53$R$NG4 1$R$NM51$R$N#PUT AX [C] $R$NM52$R$N#CALL AX [C,8,3]$R$NM54$R$N',
																	'G100 A1000$R$NM50$R$NM53$R$NG4 1$R$NM51$R$N#PUT AX [A] $R$NM52$R$N#CALL AX [A,9,4]$R$NM54$R$N',
																	''];//Measurement MDI String

END_VAR

HLI3_Init(); 
M_WarningMonitor();
M_AlarmMonitor();

(* Call CNC related code only if the HLI has been initialized succesfully! *)
IF CNCSystem.bHLIInit THEN
	M_AxesHandler();    	
	M_ManualMode(_Chan:= _SelectedChannel);
	M_ChannelHandler();	
	M_VariableViewer();	
	M_Selections(_Chan:= _SelectedChannel);	
	M_Spindle(_Chan:= _SelectedChannel);
	M_ToolHandler(_Chan:= _SelectedChannel);
	M_Homing(_Chan:= _SelectedChannel);
END_IF

{attribute 'monitoring' := 'variable'}
PROPERTY PUBLIC Alarm : Bool
GET
Alarm := _Alarm;
END_GET
END_PROPERTY

{attribute 'monitoring' := 'variable'}
PROPERTY PUBLIC AlarmMute : BOOL
SET
AlarmMute := _AlarmMute;
END_SET
END_PROPERTY

{attribute 'monitoring' := 'variable'}
PROPERTY PUBLIC AutoHome : Bool
SET
_AutoHome := AutoHome;
END_SET
END_PROPERTY

{attribute 'monitoring' := 'variable'}
PROPERTY PUBLIC AxisEnabled : Bool
GET
AxisEnabled := _AxisEnabled;
END_GET
END_PROPERTY

{attribute 'monitoring' := 'variable'}
PROPERTY PUBLIC Description : String[40]
GET
Description := _Description;
END_GET
SET
_Description := Description;
END_SET
END_PROPERTY

{attribute 'monitoring' := 'variable'}
PROPERTY PUBLIC Fault : Bool
SET
_Fault := Fault;
END_SET
END_PROPERTY

{attribute 'monitoring' := 'variable'}
PROPERTY PUBLIC FaultTimer_ET : real
GET
FaultTimer_ET := _FaultTimer_ET;
END_GET
END_PROPERTY

{attribute 'monitoring' := 'variable'}
PROPERTY PUBLIC FaultTimer_PT : real
GET
FaultTimer_PT := _FaultTimer_PT;
END_GET
SET
_FaultTimer_PT := FaultTimer_PT;
END_SET
END_PROPERTY

PROPERTY PUBLIC FeedOverride : UINT
GET
FeedOverride:= _FeedOverride;
END_GET
SET
_FeedOverride:= FeedOverride;
END_SET
END_PROPERTY

PROPERTY PUBLIC HandwheelSelected : BOOL
GET
HandwheelSelected:= (_MachineMode[0].ManualMode.nManualTyp = 1);
END_GET
END_PROPERTY

{attribute 'monitoring' := 'variable'}
PROPERTY PUBLIC Homed : Bool
GET
Homed := _Homed;
END_GET
END_PROPERTY

METHOD PRIVATE M_AlarmMonitor
VAR_INPUT
END_VAR
VAR_INST // added by the converter: edge detectors and wires of the graphical bodies
    _w1, _w2, _w3, _w4, _w5 : BOOL;
    _rt1 : R_TRIG;
END_VAR
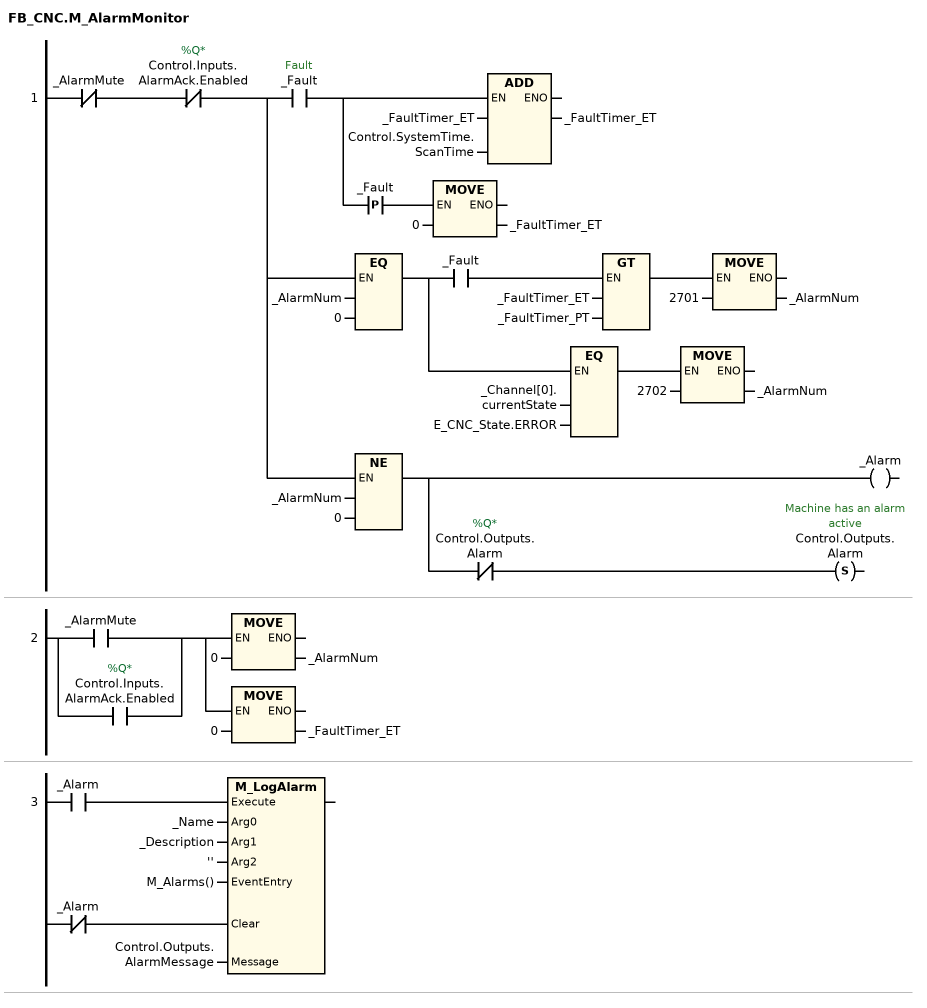
// NETWORK 1
//   Control.Inputs.AlarmAck.Enabled: AT %Q*
//   _Fault: Fault
//   _FaultTimer_ET: Fault timer elapsed
//   Control.SystemTime.ScanTime: Last scan time (Seconds)
//   _FaultTimer_PT: Fault timer preset time
//   Control.Outputs.Alarm: AT %Q* | Machine has an alarm active
_w1 := NOT _AlarmMute AND NOT Control.Inputs.AlarmAck.Enabled;
_w2 := _w1 AND _Fault;
IF _w2 THEN _FaultTimer_ET := _FaultTimer_ET + Control.SystemTime.ScanTime; END_IF
_rt1(CLK := _Fault);
IF _w2 AND _rt1.Q THEN _FaultTimer_ET := 0; END_IF
_w3 := _w1 AND _AlarmNum = 0;
IF _w3 AND _Fault AND _FaultTimer_ET > _FaultTimer_PT THEN _AlarmNum := 2701; END_IF
IF _w3 AND _Channel[0].currentState = E_CNC_State.ERROR THEN _AlarmNum := 2702; END_IF
_w4 := _w1 AND _AlarmNum <> 0;
_Alarm := _w4;
Control.Outputs.Alarm S= _w4 AND NOT Control.Outputs.Alarm;

// NETWORK 2
//   Control.Inputs.AlarmAck.Enabled: AT %Q*
//   _FaultTimer_ET: Fault timer elapsed
_w5 := _AlarmMute OR Control.Inputs.AlarmAck.Enabled;
IF _w5 THEN _AlarmNum := 0; END_IF
IF _w5 THEN _FaultTimer_ET := 0; END_IF

// NETWORK 3
M_LogAlarm(Execute := _Alarm, Arg0 := _Name, Arg1 := _Description, Arg2 := '', EventEntry := M_Alarms(), Clear := NOT _Alarm, Message := Control.Outputs.AlarmMessage);
END_METHOD

METHOD PRIVATE M_Alarms : TcEventEntry
VAR_INPUT
END_VAR
CASE _AlarmNum OF
	2701: M_Alarms:= TC_Events.TcCnc.A_2701;//Alarm	
	2702: M_Alarms:= TC_Events.TcCnc.A_2702;//Mode Error					
ELSE
	M_Alarms:= TC_Events.TcCnc.A_Undefined;
END_CASE
END_METHOD

METHOD PRIVATE M_AxesHandler
VAR_INST
	{attribute 'tc_no_symbol'}
	_HliAxisIdx					: INT;				//Loop index	
	{attribute 'tc_no_symbol'}			
	_FirstSpindle				: INT := -1;		//Spindle HLI index
	{attribute 'tc_no_symbol'}
	_fbAxesError 				: FB_AxesError;		//Axes error
END_VAR
_fbAxesError(bReset := (_Alarm AND Control.Inputs.AlarmAck.Enabled));
_AxisEnabled := TRUE;   
FOR _HliAxisIdx := 0 TO UDINT_TO_INT(gNrAx-1) DO			
	_Axis[_HliAxisIdx](bCalibrationCam:= CalibrationCam[_HliAxisIdx],
		bEnable	:= _AutoEn,
		nLogAxisNo := LogAxisNo[_HliAxisIdx]);
	_Axis[_HliAxisIdx].stOptions.bProbingSignal:= CalibrationCam[_HliAxisIdx];
		
	IF _HliAxisIdx <= UDINT_TO_INT(gNrAx-2) THEN
		_AxisNames[_HliAxisIdx] := gpCh[0]^.bahn_state.coord_r[_HliAxisIdx].axis_name_r.zeichen;
		_AxisInManual[_HliAxisIdx] := _MachineMode[0].ManualMode.nLogAxisNumber = INT_TO_UINT(_Axis[_HliAxisIdx].nLogAxisNo);
		_Axis[_HliAxisIdx].stOptions.bProbingSignal := CalibrationCam[_HliAxisIdx];	
		IF (NOT _Axis[_HliAxisIdx].stStatus.bIsEnabled) THEN    // if one axis status is "not enabled" -> reset PLCStatusAxisEnabled
			_AxisEnabled := FALSE;
		END_IF
	END_IF
		
		IF HLI3_CheckAxisValid(_HliAxisIdx) THEN
			IF _FirstSpindle = -1 AND gpAx[_HliAxisIdx]^.ipo_state.spindle_axis_r THEN  (* store HLIIndex of first spindle *)
				_FirstSpindle := _HliAxisIdx;
			END_IF
		END_IF
		
END_FOR
END_METHOD

METHOD M_ChannelHandler
VAR_INST
	{attribute 'tc_no_symbol'}
	_Chan					: INT;								//Channel index
	{attribute 'tc_no_symbol'}
	_OldSelectedChannel		: UDINT;							//Previous channel index
	{attribute 'tc_no_symbol'}
	_stOptions				: ST_CNC_CH_Options;				//HLI options for structure 
	{attribute 'tc_no_symbol'}
	_ChannelSignals			: ST_ChannelSignals;				//HLI channel signal structure
	{attribute 'tc_no_symbol'}
	_BlockSearch			: ARRAY[0..3] OF HLI3_BlockSearch;	//HLI block search structure
	{attribute 'tc_no_symbol'}
	_ErrorHandler			: ARRAY[0..3] OF FB_ChannelError;	//HLI channel error structure				
END_VAR
IF (_OldSelectedChannel <>INT_TO_UDINT(_SelectedChannel)) THEN
	_ChannelSignals.SingleBlock 		:= _MachineMode[_SelectedChannel].ChannelSignals.SingleBlock;
	_ChannelSignals.PrgBlockIgnore		:= _MachineMode[_SelectedChannel].ChannelSignals.PrgBlockIgnore;
	_ChannelSignals.M01Stop 			:= _MachineMode[_SelectedChannel].ChannelSignals.M01Stop;
	_ChannelSignals.Backward 			:= _MachineMode[_SelectedChannel].ChannelSignals.Backward;
	_ChannelSignals.FeedHold 			:= _MachineMode[_SelectedChannel].ChannelSignals.FeedHold;
	_OldSelectedChannel 				:= INT_TO_UDINT(_SelectedChannel);
END_IF

_MachineMode[_SelectedChannel].ChannelSignals.SingleBlock 	:= _ChannelSignals.SingleBlock;
_MachineMode[_SelectedChannel].ChannelSignals.PrgBlockIgnore:= _ChannelSignals.PrgBlockIgnore;
_MachineMode[_SelectedChannel].ChannelSignals.M01Stop 		:= _ChannelSignals.M01Stop;
_MachineMode[_SelectedChannel].ChannelSignals.Backward 		:= _ChannelSignals.Backward;
_MachineMode[_SelectedChannel].ChannelSignals.FeedHold 		:= _ChannelSignals.FeedHold;

_stOptions.bReferenceModeStartRequired := FALSE;
//_stOptions.bDisableCNCPLCWatchDog := TRUE;

FOR _Chan := 0 TO MaxChannelIdx DO
	IF (HLI3_CheckChannelValid(_Chan)) THEN		
		
		_MachineMode[_Chan].Mode 	:= _Channel[_Chan].currentMode;
		_MachineMode[_Chan].State	:= _Channel[_Chan].currentState;
		_ErrorHandler[_Chan](nChanIdx	:= _Chan);				

		_Channel[_Chan]
			(nChanIdx			:= _Chan,							
			 bModeStandby		:= _MachineMode[_Chan].Standby,
			 bModeAutomatic		:= _MachineMode[_Chan].Automatic,
			 bModeManual		:= _MachineMode[_Chan].Manual,
			 bModeMDI			:= _MachineMode[_Chan].MDI,	 
			 bModeReference		:= _MachineMode[_Chan].Homing,
			 bStateSelect		:= _MachineMode[_Chan].Select,
			 bStateReady		:= _MachineMode[_Chan].Ready,
			 bStateStart		:= _MachineMode[_Chan].Start,
			 bStateStop			:= _MachineMode[_Chan].Stop,
			 bStateReset		:= _MachineMode[_Chan].Reset,
			 nFeedOverride		:= _FeedOverride * 10,
			 nRapidFeedOverride := _FeedOverride * 10, 
			 sProgramName		:= _MachineMode[_Chan].ProgramName,			 
			 sMDIString			:= _MachineMode[_Chan].MDIString,
			 bBackwardMotion	:= _MachineMode[_Chan].ChannelSignals.Backward,
			 bPrgBlockIgnore	:= _MachineMode[_Chan].ChannelSignals.PrgBlockIgnore,
			 bFeedHold			:= _MachineMode[_Chan].ChannelSignals.FeedHold,
			 bSingleBlock		:= _MachineMode[_Chan].ChannelSignals.SingleBlock,
			 bDoSingleBlock		:= _MachineMode[_Chan].ChannelSignals.DoSingleBlock,
			 bM01Stop			:= _MachineMode[_Chan].ChannelSignals.M01Stop,
			 nSyntaxCheck		:= _MachineMode[_Chan].SyntaxCheck.nType,
			 bM30Acknowledgement:= TRUE,
			 stManualModeParameter  	 	 := stManualModeParameter[_Chan],
			 stManualModeControlElements	 := stManualModeControlElements[_Chan],
			 stManualModeControlElementState := stManualModeControlElementState,
			 stOptions			:= 	_stOptions
			);
			
		_r_trig[_Chan](CLK:= gpCh[_Chan]^.bahn_state.program_end_r);
		_ProgramEnd[_Chan]:= _r_trig[_Chan].Q;
		
		_BlockSearch[_Chan]
			(nChanIdx			:= _Chan,
			 bStartRead      	:= _MachineMode[_Chan].BlockSearch.bStartRead,   (* Edge signal *)
			 bStartWrite     	:= _MachineMode[_Chan].BlockSearch.bStartWrite,  (* Edge signal *)
			 BlockSearch		:= _MachineMode[_Chan].BlockSearch
			);
		
		CNCSystem.Channel[_Chan].ActDistance 	:= DINT_TO_LREAL(_BlockSearch[_Chan].coveredDistance_AfterReset) / 10.0;
		CNCSystem.Channel[_Chan].ActBlockCount 	:= _BlockSearch[_Chan].actualBlockCount_AfterReset;
						
	END_IF
END_FOR

_CurrentNCProgram := gpCh[0]^.bahn_state.file_name_r.zeichen;
_CurrentLine:= gpCh[0]^.bahn_state.block_nr_r;
END_METHOD

METHOD PRIVATE M_Homing
VAR_INPUT
	{attribute 'tc_no_symbol'}
	_Chan								 : INT;									//Channel index
END_VAR
VAR_INST
	{attribute 'tc_no_symbol'}
	_Step                  			 	 : ARRAY[0..3] OF INT;					//Step counter
	{attribute 'tc_no_symbol'}
	_Axe					 			 : UINT;								//Axes index
	{attribute 'tc_no_symbol'}
	_SetDrivePosition					 : BOOL;								//Set drive position
	{attribute 'tc_no_symbol'}
	_DeleteDrivePosition				 : BOOL;								//Delete drive position
	{attribute 'tc_no_symbol'}	
	_fb_CNCAX5000SetPositionOffset		 : FB_CNCAX5000SetPositionOffset;		//Sets encoder position in drive memory
	{attribute 'tc_no_symbol'}
	_fb_CNCAX5000DeletePositionOffset	 : FB_CNCAX5000DeletePositionOffset;	//Clears drive memory
END_VAR
IF _MachineMode[_Chan].State = E_CNC_State.ERROR OR Control.PackMLState.Stopped THEN
   _Step[_Chan] := 0;
END_IF
 
CASE _Referencing OF

//Homing Method with Calibration Cam. This method uses the Position Offsets stored in the CNC Params. The encoder position is NOT stored in memory.
E_CNC_HomingMethod.Homing:

	CASE _Step[_Chan] OF
		0: //Idle
			IF _AutoHome AND NOT _Alarm THEN
				_Homed := FALSE;
				_Axe:=0;
			    _Step[_Chan] := 1;
			ELSIF _ManHome.Queued AND NOT _Alarm THEN
				_Homed := FALSE;
				IF _ManHome.Enabled THEN
					_Axe:=INT_TO_UINT(_SelectedAxis);
					_Step[_Chan] := 10;
				END_IF
			END_IF
		
		1://Update Homing Offsets
			_Axis[0].fRefOffset:= _PositionOffset[0];
			_Axis[0].bSetRefOffset:= TRUE;
			_Axis[1].fRefOffset:= _PositionOffset[1];
			_Axis[1].bSetRefOffset:= TRUE;
			_Axis[2].fRefOffset:= _PositionOffset[2];
			_Axis[2].bSetRefOffset:= TRUE;
			_Axis[3].fRefOffset:= _PositionOffset[3];
			_Axis[3].bSetRefOffset:= TRUE;
			_Axis[4].fRefOffset:= _PositionOffset[4];
			_Axis[4].bSetRefOffset:= TRUE;

			_Step[_Chan] := 2;
	
	
		2://Enable Homing
			_MachineMode[0].Homing:= TRUE;

			IF _Axis[0].stStatus.bHomingDone AND _Axis[1].stStatus.bHomingDone AND 
				_Axis[2].stStatus.bHomingDone AND _Axis[3].stStatus.bHomingDone AND _Axis[4].stStatus.bHomingDone THEN
					_Step[_Chan] := 3;
			END_IF
	
		3: //Wait for CNC to reach park positions
		 	IF _MachineMode[_Chan].State = E_CNC_State.READY THEN
		     	_Step[_Chan] := 4;
		 	END_IF
		
		4://Set mode to standby	
			_Homed := TRUE;
			_MachineMode[_Chan].Standby := TRUE;
			IF NOT _Autohome AND NOT _ManHome.Enabled AND _MachineMode[_Chan].Mode = E_CNC_Mode.STANDBY_MODE THEN
				_Step[_Chan] := 0;
			END_IF
			
		//Single Axis Manual Home
		10://Set MDI Mode
			_MachineMode[_Chan].MDI := TRUE;
			IF _MachineMode[_Chan].Mode = E_CNC_Mode.MDI_MODE THEN
				_Step[_Chan] := 11;
	    	END_IF
			
		11://Set homing string for indiviudal axis
			CASE _Axe OF
				0: _MachineMode[_Chan].MDIString := 'G74 X0';
				1: _MachineMode[_Chan].MDIString := 'G74 Y0';
				2: _MachineMode[_Chan].MDIString := 'G74 Z0';
				3: _MachineMode[_Chan].MDIString := 'G74 C0';
				4: _MachineMode[_Chan].MDIString := 'G74 A0';
			END_CASE
			_MachineMode[_Chan].Start := TRUE;
			_SetDrivePosition := FALSE;
	 		_Step[_Chan] := 12;
			
		12://Wait for CNC ready state
			IF _MachineMode[_Chan].State = E_CNC_State.READY THEN
	       		_Step[_Chan] := 13;
	    	END_IF
			
		13://Park Axis
			_MachineMode[_Chan].MDIString := CONCAT(_AxisNames[_SelectedAxis],TO_STRING(_ParkPositions[_SelectedAxis]));
			_MachineMode[_Chan].Start := TRUE;
			_Step[_Chan] := 14;
		
		14: //Wait for CNC to start moving to park positions
		 	IF _MachineMode[_Chan].State = E_CNC_State.ACTIVE THEN
		     	_Step[_Chan] := 15;
		 	END_IF		
			
		15: //Wait for CNC to reach park positions
		 	IF _MachineMode[_Chan].State = E_CNC_State.READY THEN
		     	_Step[_Chan] := 16;
		 	END_IF
		
		16://Set mode to standby	
			_Homed := TRUE;
			_MachineMode[_Chan].Standby := TRUE;
			IF NOT _Autohome AND NOT _ManHome.Enabled AND _MachineMode[_Chan].Mode = E_CNC_Mode.STANDBY_MODE THEN
				_Step[_Chan] := 0;
			END_IF
	END_CASE		


//Measurement Method With Probing Signal. This method uses the Position Offsets stored in the PLC. The encoder position IS stored in memory.
E_CNC_HomingMethod.Measurment:

	CASE _Step[_Chan] OF
		0: //Idle
			IF _AutoHome AND NOT _Alarm THEN
				_SetDrivePosition := FALSE;
				FOR _Axe := 0 TO UDINT_TO_UINT(gNrAx-2) DO
					_Axis[_MeasurementOrder[_Axe]].bSetRefOffset := FALSE;
					_Axis[_MeasurementOrder[_Axe]].stOptions.bResetCalibration := TRUE;
				END_FOR;
				_Homed := FALSE;
				_Axe:= 0;
			    _Step[_Chan] := 1;
			ELSIF _ManHome.Queued AND NOT _Alarm THEN
				_Homed := FALSE;
				IF _ManHome.Enabled THEN
					_Axe:=INT_TO_UINT(_SelectedAxis);
					_Step[_Chan] := 1;
				END_IF
			END_IF
			
		1://Enable Axes and set Standby Mode
			_AutoEn := TRUE;
			_MachineMode[_Chan].Standby := TRUE;
			IF _AxisEnabled AND _MachineMode[_Chan].Mode = E_CNC_Mode.STANDBY_MODE THEN
				_Step[_Chan] := 2;
			END_IF
	    	
	    2: //Set MDI mode
			_MachineMode[_Chan].MDI := TRUE;
			IF _MachineMode[_Chan].Mode = E_CNC_Mode.MDI_MODE THEN
				_Step[_Chan] := 3;
	    	END_IF
			
		3: //Reset homing done bool to allow ignorance of software limits
			IF _Axis[_MeasurementOrder[_Axe]].stStatus.bHomingDone = FALSE THEN
				_Axis[_MeasurementOrder[_Axe]].stOptions.bResetCalibration := FALSE;	
				_Step[_Chan] := 4;
			END_IF
			
	    4: //Create homing MDI string
			IF _ManHome.Enabled THEN
				_MachineMode[_Chan].MDIString := _MeasurementMDIString[_Axe];
			ELSE
				_MachineMode[_Chan].MDIString := _MeasurementMDIString[_MeasurementOrder[_Axe]];	
			END_IF
			_MachineMode[_Chan].Start := TRUE;
			_SetDrivePosition := FALSE;
	 		_Step[_Chan] := 5;
		
	    5: //Wait for CNC to start moving to home positions
	    	IF _MachineMode[_Chan].State = E_CNC_State.ACTIVE THEN
	       		_Step[_Chan] := 6;
	    	END_IF	
	
		6://Wait for CNC to reach home positions
		
				//M50 Clear Reference Flag
				IF CNCSystem.Channel[0].M[50].bState_rw THEN
					_Axis[_MeasurementOrder[_Axe]].stOptions.bResetCalibration := TRUE;
					IF _Axis[_MeasurementOrder[_Axe]].stStatus.bHomingDone = FALSE THEN
						_Axis[_MeasurementOrder[_Axe]].stOptions.bResetCalibration := FALSE;
						CNCSystem.Channel[0].M[50].bState_rw := FALSE;
					END_IF
				END_IF
				
				//M51 Set Drive Position
				IF CNCSystem.Channel[0].M[51].bState_rw THEN
					_SetDrivePosition := TRUE;
				END_IF
				IF _Axis[_MeasurementOrder[_Axe]].stStatus.fActPosACS > (_PositionOffset[_MeasurementOrder[_Axe]] -1) AND  _Axis[_MeasurementOrder[_Axe]].stStatus.fActPosACS < (_PositionOffset[_MeasurementOrder[_Axe]] +1) THEN
					CNCSystem.Channel[0].M[51].bState_rw := FALSE;
					_SetDrivePosition := FALSE;
				END_IF 
				
				//M52 Set Axis as Homed
				IF CNCSystem.Channel[0].M[52].bState_rw THEN
					_Axis[_MeasurementOrder[_Axe]].fRefOffset := 0;
					_Axis[_MeasurementOrder[_Axe]].bSetRefOffset := TRUE;
					IF _Axis[_MeasurementOrder[_Axe]].stStatus.bHomingDone = TRUE THEN
						CNCSystem.Channel[0].M[52].bState_rw := FALSE;
						_Axis[_MeasurementOrder[_Axe]].bSetRefOffset := FALSE;
					END_IF
				END_IF
				
				//M53 Disable Axis
				IF CNCSystem.Channel[0].M[53].bState_rw THEN
					_AutoEn := FALSE;
					IF NOT _Axis[_MeasurementOrder[_Axe]].stStatus.bIsEnabled THEN
						CNCSystem.Channel[0].M[53].bState_rw := FALSE;
					END_IF
				END_IF
				
				//M54 Enable Axis
				IF CNCSystem.Channel[0].M[54].bState_rw THEN
					_AutoEn := TRUE;
					IF _Axis[_MeasurementOrder[_Axe]].stStatus.bIsEnabled THEN
						CNCSystem.Channel[0].M[54].bState_rw := FALSE;
						_Step[_Chan] := 7;	
					END_IF
				END_IF
				
	    7: //Wait for CNC to be Ready
	    	IF _MachineMode[_Chan].State = E_CNC_State.READY THEN
	       		IF (_ManHome.Enabled OR _Axe >= (gNrAx-3)) THEN//)>= 1 THEN
					_Step[_Chan] := 8;
				ELSE
					_Axe:=_Axe+1;
					_Step[_Chan] := 3;
				END_IF
	    	END_IF	
				
		8://Create parking MDI string
			IF _ManHome.Enabled THEN
				_ParkMDIString := CONCAT(_AxisNames[_SelectedAxis],TO_STRING(_ParkPositions[_SelectedAxis]));
			ELSE	
				FOR _Axe := 0 TO UDINT_TO_UINT(gNrAx-2) BY 1 DO	
					IF _Axe = 0 THEN
						_ParkMDIString	:= concat(_AxisNames[_Axe],TO_STRING(_ParkPositions[_Axe]));
					ELSE
						_ParkMDIString	:= concat(_ParkMDIString,concat(' ', concat(_AxisNames[_Axe],TO_STRING(_ParkPositions[_Axe]))));
					END_IF
				END_FOR	
			END_IF
			_MachineMode[_Chan].MDIString := _ParkMDIString;
			_MachineMode[_Chan].Start := TRUE;
			_Step[_Chan] := 9;
		
		9: //Wait for CNC to start moving to park positions
		 	IF _MachineMode[_Chan].State = E_CNC_State.ACTIVE THEN
		     	_Step[_Chan] := 10;
		 	END_IF		
			
		10: //Wait for CNC to reach park positions
		 	IF _MachineMode[_Chan].State = E_CNC_State.READY THEN
		     	_Step[_Chan] := 11;
		 	END_IF
		
		11://Set mode to standby	
			_Homed := TRUE;
			_MachineMode[_Chan].Standby := TRUE;
			IF NOT _Autohome AND NOT _ManHome.Enabled AND _MachineMode[_Chan].Mode = E_CNC_Mode.STANDBY_MODE THEN
				_Step[_Chan] := 0;
			END_IF
			
	END_CASE

END_CASE

//Delete Position Offset
_fb_CNCAX5000DeletePositionOffset(nLogAxisNo:= TO_UINT(_Axis[_MeasurementOrder[_Axe]].nLogAxisNo), Execute:= _DeleteDrivePosition, Memory:= tc3_cnc_drive.E_PositionOffsetMemory.ePositionOffsetMemory_Drive);

//Set Position Offset
_fb_CNCAX5000SetPositionOffset(nLogAxisNo:= TO_UINT(_Axis[_MeasurementOrder[_Axe]].nLogAxisNo), Execute:= _SetDrivePosition, Position:= _PositionOffset[_MeasurementOrder[_Axe]], Memory:= tc3_cnc_drive.E_PositionOffsetMemory.ePositionOffsetMemory_Drive);
END_METHOD

METHOD PRIVATE M_ManualMode
VAR_INPUT
	{attribute 'tc_no_symbol'}
	_Chan								 : INT;									//Channel index
END_VAR	
VAR_INST
	{attribute 'tc_no_symbol'}
	_fbUintUdInt						 : ARRAY [0..3] OF FB_Uint_Udint;		//Uint to udint FB
	{attribute 'tc_no_symbol'}
	_HandWheelBig						 : UDINT;								//Handwheel value
END_VAR
IF (HLI3_CheckChannelValid(_Chan)) THEN

	stManualModeParameter[_Chan].stChannelParameter.nChanIdx := _Chan;       (* Channel 1 *)
	stManualModeParameter[_Chan].stChannelParameter.nInc := _MachineMode[_Chan].ManualMode.nInc * 10;
	stManualModeParameter[_Chan].stChannelParameter.bG200ConfigurationViaPLC := TRUE;		
	
	stManualModeParameter[_Chan].stChannelParameter.eManualType := UINT_TO_INT(_MachineMode[_Chan].ManualMode.nManualTyp);			
	IF (stManualModeParameter[_Chan].stChannelParameter.eManualType = E_CNC_ManualType.Handwheel AND _Chan <> _SelectedChannel) THEN	(* if in Handwheel mode and the channel is NOT selected -> leave handwheel mode and change to TippMode*)
		stManualModeParameter[_Chan].stChannelParameter.eManualType := E_CNC_ManualType.TippMode;
	END_IF		
	
